//     PlcTask Inputs/GVL_iXlinker.EtherCAT_Master_EJxxxx.Beckhoff_EJ3xxx.A_0005_EJ3058_0000_0020.AI_Standard_Channel_3.Status/Limit_2 <-> AI Standard Channel 3/Status/Limit 2
//     PlcTask Inputs/GVL_iXlinker.EtherCAT_Master_EJxxxx.Beckhoff_EJ3xxx.A_0005_EJ3058_0000_0020.AI_Standard_Channel_4.Status/Limit_1 <-> AI Standard Channel 4/Status/Limit 1
//     PlcTask Inputs/GVL_iXlinker.EtherCAT_Master_EJxxxx.Beckhoff_EJ3xxx.A_0005_EJ3058_0000_0020.AI_Standard_Channel_4.Status/Limit_2 <-> AI Standard Channel 4/Status/Limit 2
//     PlcTask Inputs/GVL_iXlinker.EtherCAT_Master_EJxxxx.Beckhoff_EJ3xxx.A_0005_EJ3058_0000_0020.AI_Standard_Channel_5.Status/Limit_1 <-> AI Standard Channel 5/Status/Limit 1
//     PlcTask Inputs/GVL_iXlinker.EtherCAT_Master_EJxxxx.Beckhoff_EJ3xxx.A_0005_EJ3058_0000_0020.AI_Standard_Channel_5.Status/Limit_2 <-> AI Standard Channel 5/Status/Limit 2
//     PlcTask Inputs/GVL_iXlinker.EtherCAT_Master_EJxxxx.Beckhoff_EJ3xxx.A_0005_EJ3058_0000_0020.AI_Standard_Channel_6.Status/Limit_1 <-> AI Standard Channel 6/Status/Limit 1
//     PlcTask Inputs/GVL_iXlinker.EtherCAT_Master_EJxxxx.Beckhoff_EJ3xxx.A_0005_EJ3058_0000_0020.AI_Standard_Channel_6.Status/Limit_2 <-> AI Standard Channel 6/Status/Limit 2
//     PlcTask Inputs/GVL_iXlinker.EtherCAT_Master_EJxxxx.Beckhoff_EJ3xxx.A_0005_EJ3058_0000_0020.AI_Standard_Channel_7.Status/Limit_1 <-> AI Standard Channel 7/Status/Limit 1
//     PlcTask Inputs/GVL_iXlinker.EtherCAT_Master_EJxxxx.Beckhoff_EJ3xxx.A_0005_EJ3058_0000_0020.AI_Standard_Channel_7.Status/Limit_2 <-> AI Standard Channel 7/Status/Limit 2
//     PlcTask Inputs/GVL_iXlinker.EtherCAT_Master_EJxxxx.Beckhoff_EJ3xxx.A_0005_EJ3058_0000_0020.AI_Standard_Channel_8.Status/Limit_1 <-> AI Standard Channel 8/Status/Limit 1
//     PlcTask Inputs/GVL_iXlinker.EtherCAT_Master_EJxxxx.Beckhoff_EJ3xxx.A_0005_EJ3058_0000_0020.AI_Standard_Channel_8.Status/Limit_2 <-> AI Standard Channel 8/Status/Limit 2
//     PlcTask Inputs/GVL_iXlinker.EtherCAT_Master_EJxxxx.Beckhoff_EJ3xxx.A_0005_EJ3058_0000_0020.AI_Standard_Channel_1.Status/Error <-> AI Standard Channel 1/Status/Error
//     PlcTask Inputs/GVL_iXlinker.EtherCAT_Master_EJxxxx.Beckhoff_EJ3xxx.A_0005_EJ3058_0000_0020.AI_Standard_Channel_2.Status/Error <-> AI Standard Channel 2/Status/Error
//     PlcTask Inputs/GVL_iXlinker.EtherCAT_Master_EJxxxx.Beckhoff_EJ3xxx.A_0005_EJ3058_0000_0020.AI_Standard_Channel_3.Status/Error <-> AI Standard Channel 3/Status/Error
//     PlcTask Inputs/GVL_iXlinker.EtherCAT_Master_EJxxxx.Beckhoff_EJ3xxx.A_0005_EJ3058_0000_0020.AI_Standard_Channel_4.Status/Error <-> AI Standard Channel 4/Status/Error
//     PlcTask Inputs/GVL_iXlinker.EtherCAT_Master_EJxxxx.Beckhoff_EJ3xxx.A_0005_EJ3058_0000_0020.AI_Standard_Channel_5.Status/Error <-> AI Standard Channel 5/Status/Error
//     PlcTask Inputs/GVL_iXlinker.EtherCAT_Master_EJxxxx.Beckhoff_EJ3xxx.A_0005_EJ3058_0000_0020.AI_Standard_Channel_6.Status/Error <-> AI Standard Channel 6/Status/Error
//     PlcTask Inputs/GVL_iXlinker.EtherCAT_Master_EJxxxx.Beckhoff_EJ3xxx.A_0005_EJ3058_0000_0020.AI_Standard_Channel_7.Status/Error <-> AI Standard Channel 7/Status/Error
//     PlcTask Inputs/GVL_iXlinker.EtherCAT_Master_EJxxxx.Beckhoff_EJ3xxx.A_0005_EJ3058_0000_0020.AI_Standard_Channel_8.Status/Error <-> AI Standard Channel 8/Status/Error
//     PlcTask Inputs/GVL_iXlinker.EtherCAT_Master_EJxxxx.Beckhoff_EJ3xxx.A_0005_EJ3058_0000_0020.AI_Standard_Channel_1.Status/TxPDO_State <-> AI Standard Channel 1/Status/TxPDO State
//     PlcTask Inputs/GVL_iXlinker.EtherCAT_Master_EJxxxx.Beckhoff_EJ3xxx.A_0005_EJ3058_0000_0020.AI_Standard_Channel_2.Status/TxPDO_State <-> AI Standard Channel 2/Status/TxPDO State
//     PlcTask Inputs/GVL_iXlinker.EtherCAT_Master_EJxxxx.Beckhoff_EJ3xxx.A_0005_EJ3058_0000_0020.AI_Standard_Channel_3.Status/TxPDO_State <-> AI Standard Channel 3/Status/TxPDO State
//     PlcTask Inputs/GVL_iXlinker.EtherCAT_Master_EJxxxx.Beckhoff_EJ3xxx.A_0005_EJ3058_0000_0020.AI_Standard_Channel_4.Status/TxPDO_State <-> AI Standard Channel 4/Status/TxPDO State
//     PlcTask Inputs/GVL_iXlinker.EtherCAT_Master_EJxxxx.Beckhoff_EJ3xxx.A_0005_EJ3058_0000_0020.AI_Standard_Channel_5.Status/TxPDO_State <-> AI Standard Channel 5/Status/TxPDO State
//     PlcTask Inputs/GVL_iXlinker.EtherCAT_Master_EJxxxx.Beckhoff_EJ3xxx.A_0005_EJ3058_0000_0020.AI_Standard_Channel_6.Status/TxPDO_State <-> AI Standard Channel 6/Status/TxPDO State
//     PlcTask Inputs/GVL_iXlinker.EtherCAT_Master_EJxxxx.Beckhoff_EJ3xxx.A_0005_EJ3058_0000_0020.AI_Standard_Channel_7.Status/TxPDO_State <-> AI Standard Channel 7/Status/TxPDO State
//     PlcTask Inputs/GVL_iXlinker.EtherCAT_Master_EJxxxx.Beckhoff_EJ3xxx.A_0005_EJ3058_0000_0020.AI_Standard_Channel_8.Status/TxPDO_State <-> AI Standard Channel 8/Status/TxPDO State
//     PlcTask Inputs/GVL_iXlinker.EtherCAT_Master_EJxxxx.Beckhoff_EJ3xxx.A_0005_EJ3058_0000_0020.AI_Standard_Channel_1.Status/TxPDO_Toggle <-> AI Standard Channel 1/Status/TxPDO Toggle
//     PlcTask Inputs/GVL_iXlinker.EtherCAT_Master_EJxxxx.Beckhoff_EJ3xxx.A_0005_EJ3058_0000_0020.AI_Standard_Channel_2.Status/TxPDO_Toggle <-> AI Standard Channel 2/Status/TxPDO Toggle
//     PlcTask Inputs/GVL_iXlinker.EtherCAT_Master_EJxxxx.Beckhoff_EJ3xxx.A_0005_EJ3058_0000_0020.AI_Standard_Channel_3.Status/TxPDO_Toggle <-> AI Standard Channel 3/Status/TxPDO Toggle
//     PlcTask Inputs/GVL_iXlinker.EtherCAT_Master_EJxxxx.Beckhoff_EJ3xxx.A_0005_EJ3058_0000_0020.AI_Standard_Channel_4.Status/TxPDO_Toggle <-> AI Standard Channel 4/Status/TxPDO Toggle
//     PlcTask Inputs/GVL_iXlinker.EtherCAT_Master_EJxxxx.Beckhoff_EJ3xxx.A_0005_EJ3058_0000_0020.AI_Standard_Channel_5.Status/TxPDO_Toggle <-> AI Standard Channel 5/Status/TxPDO Toggle
//     PlcTask Inputs/GVL_iXlinker.EtherCAT_Master_EJxxxx.Beckhoff_EJ3xxx.A_0005_EJ3058_0000_0020.AI_Standard_Channel_6.Status/TxPDO_Toggle <-> AI Standard Channel 6/Status/TxPDO Toggle
//     PlcTask Inputs/GVL_iXlinker.EtherCAT_Master_EJxxxx.Beckhoff_EJ3xxx.A_0005_EJ3058_0000_0020.AI_Standard_Channel_7.Status/TxPDO_Toggle <-> AI Standard Channel 7/Status/TxPDO Toggle
//     PlcTask Inputs/GVL_iXlinker.EtherCAT_Master_EJxxxx.Beckhoff_EJ3xxx.A_0005_EJ3058_0000_0020.AI_Standard_Channel_8.Status/TxPDO_Toggle <-> AI Standard Channel 8/Status/TxPDO Toggle
//     PlcTask Inputs/GVL_iXlinker.EtherCAT_Master_EJxxxx.Beckhoff_EJ3xxx.A_0005_EJ3058_0000_0020.AI_Standard_Channel_1.Value <-> AI Standard Channel 1/Value
//     PlcTask Inputs/GVL_iXlinker.EtherCAT_Master_EJxxxx.Beckhoff_EJ3xxx.A_0005_EJ3058_0000_0020.AI_Standard_Channel_2.Value <-> AI Standard Channel 2/Value
//     PlcTask Inputs/GVL_iXlinker.EtherCAT_Master_EJxxxx.Beckhoff_EJ3xxx.A_0005_EJ3058_0000_0020.AI_Standard_Channel_3.Value <-> AI Standard Channel 3/Value
//     PlcTask Inputs/GVL_iXlinker.EtherCAT_Master_EJxxxx.Beckhoff_EJ3xxx.A_0005_EJ3058_0000_0020.AI_Standard_Channel_4.Value <-> AI Standard Channel 4/Value
//     PlcTask Inputs/GVL_iXlinker.EtherCAT_Master_EJxxxx.Beckhoff_EJ3xxx.A_0005_EJ3058_0000_0020.AI_Standard_Channel_5.Value <-> AI Standard Channel 5/Value
//     PlcTask Inputs/GVL_iXlinker.EtherCAT_Master_EJxxxx.Beckhoff_EJ3xxx.A_0005_EJ3058_0000_0020.AI_Standard_Channel_6.Value <-> AI Standard Channel 6/Value
//     PlcTask Inputs/GVL_iXlinker.EtherCAT_Master_EJxxxx.Beckhoff_EJ3xxx.A_0005_EJ3058_0000_0020.AI_Standard_Channel_7.Value <-> AI Standard Channel 7/Value
//     PlcTask Inputs/GVL_iXlinker.EtherCAT_Master_EJxxxx.Beckhoff_EJ3xxx.A_0005_EJ3058_0000_0020.AI_Standard_Channel_8.Value <-> AI Standard Channel 8/Value
//     PlcTask Inputs/GVL_iXlinker.EtherCAT_Master_EJxxxx.Beckhoff_EJ3xxx.A_0005_EJ3058_0000_0020.WcState.WcState <-> WcState/WcState
//     PlcTask Inputs/GVL_iXlinker.EtherCAT_Master_EJxxxx.Beckhoff_EJ3xxx.A_0005_EJ3058_0000_0020.WcState.InputToggle <-> WcState/InputToggle
//     PlcTask Inputs/GVL_iXlinker.EtherCAT_Master_EJxxxx.Beckhoff_EJ3xxx.A_0005_EJ3058_0000_0020.InfoData.AdsAddr <-> InfoData/AdsAddr
//     PlcTask Inputs/GVL_iXlinker.EtherCAT_Master_EJxxxx.Beckhoff_EJ3xxx.A_0005_EJ3058_0000_0020.InfoData.State <-> InfoData/State
//   PLC/PLC Instance <-> EtherCAT Master EJxxxx/Beckhoff EJ3xxx/A_0006(EJ3068-0000-0020)
//     PlcTask Inputs/GVL_iXlinker.EtherCAT_Master_EJxxxx.Beckhoff_EJ3xxx.A_0006_EJ3068_0000_0020.AI_Standard_Channel_1.Status/Underrange <-> AI Standard Channel 1/Status/Underrange
//     PlcTask Inputs/GVL_iXlinker.EtherCAT_Master_EJxxxx.Beckhoff_EJ3xxx.A_0006_EJ3068_0000_0020.AI_Standard_Channel_2.Status/Underrange <-> AI Standard Channel 2/Status/Underrange
//     PlcTask Inputs/GVL_iXlinker.EtherCAT_Master_EJxxxx.Beckhoff_EJ3xxx.A_0006_EJ3068_0000_0020.AI_Standard_Channel_3.Status/Underrange <-> AI Standard Channel 3/Status/Underrange
//     PlcTask Inputs/GVL_iXlinker.EtherCAT_Master_EJxxxx.Beckhoff_EJ3xxx.A_0006_EJ3068_0000_0020.AI_Standard_Channel_4.Status/Underrange <-> AI Standard Channel 4/Status/Underrange
//     PlcTask Inputs/GVL_iXlinker.EtherCAT_Master_EJxxxx.Beckhoff_EJ3xxx.A_0006_EJ3068_0000_0020.AI_Standard_Channel_5.Status/Underrange <-> AI Standard Channel 5/Status/Underrange
//     PlcTask Inputs/GVL_iXlinker.EtherCAT_Master_EJxxxx.Beckhoff_EJ3xxx.A_0006_EJ3068_0000_0020.AI_Standard_Channel_6.Status/Underrange <-> AI Standard Channel 6/Status/Underrange
//     PlcTask Inputs/GVL_iXlinker.EtherCAT_Master_EJxxxx.Beckhoff_EJ3xxx.A_0006_EJ3068_0000_0020.AI_Standard_Channel_7.Status/Underrange <-> AI Standard Channel 7/Status/Underrange
//     PlcTask Inputs/GVL_iXlinker.EtherCAT_Master_EJxxxx.Beckhoff_EJ3xxx.A_0006_EJ3068_0000_0020.AI_Standard_Channel_8.Status/Underrange <-> AI Standard Channel 8/Status/Underrange
//     PlcTask Inputs/GVL_iXlinker.EtherCAT_Master_EJxxxx.Beckhoff_EJ3xxx.A_0006_EJ3068_0000_0020.AI_Standard_Channel_1.Status/Overrange <-> AI Standard Channel 1/Status/Overrange
//     PlcTask Inputs/GVL_iXlinker.EtherCAT_Master_EJxxxx.Beckhoff_EJ3xxx.A_0006_EJ3068_0000_0020.AI_Standard_Channel_2.Status/Overrange <-> AI Standard Channel 2/Status/Overrange
//     PlcTask Inputs/GVL_iXlinker.EtherCAT_Master_EJxxxx.Beckhoff_EJ3xxx.A_0006_EJ3068_0000_0020.AI_Standard_Channel_3.Status/Overrange <-> AI Standard Channel 3/Status/Overrange
//     PlcTask Inputs/GVL_iXlinker.EtherCAT_Master_EJxxxx.Beckhoff_EJ3xxx.A_0006_EJ3068_0000_0020.AI_Standard_Channel_4.Status/Overrange <-> AI Standard Channel 4/Status/Overrange
//     PlcTask Inputs/GVL_iXlinker.EtherCAT_Master_EJxxxx.Beckhoff_EJ3xxx.A_0006_EJ3068_0000_0020.AI_Standard_Channel_5.Status/Overrange <-> AI Standard Channel 5/Status/Overrange
//     PlcTask Inputs/GVL_iXlinker.EtherCAT_Master_EJxxxx.Beckhoff_EJ3xxx.A_0006_EJ3068_0000_0020.AI_Standard_Channel_6.Status/Overrange <-> AI Standard Channel 6/Status/Overrange
//     PlcTask Inputs/GVL_iXlinker.EtherCAT_Master_EJxxxx.Beckhoff_EJ3xxx.A_0006_EJ3068_0000_0020.AI_Standard_Channel_7.Status/Overrange <-> AI Standard Channel 7/Status/Overrange
//     PlcTask Inputs/GVL_iXlinker.EtherCAT_Master_EJxxxx.Beckhoff_EJ3xxx.A_0006_EJ3068_0000_0020.AI_Standard_Channel_8.Status/Overrange <-> AI Standard Channel 8/Status/Overrange
//     PlcTask Inputs/GVL_iXlinker.EtherCAT_Master_EJxxxx.Beckhoff_EJ3xxx.A_0006_EJ3068_0000_0020.AI_Standard_Channel_1.Status/Limit_1 <-> AI Standard Channel 1/Status/Limit 1
//     PlcTask Inputs/GVL_iXlinker.EtherCAT_Master_EJxxxx.Beckhoff_EJ3xxx.A_0006_EJ3068_0000_0020.AI_Standard_Channel_1.Status/Limit_2 <-> AI Standard Channel 1/Status/Limit 2
//     PlcTask Inputs/GVL_iXlinker.EtherCAT_Master_EJxxxx.Beckhoff_EJ3xxx.A_0006_EJ3068_0000_0020.AI_Standard_Channel_2.Status/Limit_1 <-> AI Standard Channel 2/Status/Limit 1
//     PlcTask Inputs/GVL_iXlinker.EtherCAT_Master_EJxxxx.Beckhoff_EJ3xxx.A_0006_EJ3068_0000_0020.AI_Standard_Channel_2.Status/Limit_2 <-> AI Standard Channel 2/Status/Limit 2
//     PlcTask Inputs/GVL_iXlinker.EtherCAT_Master_EJxxxx.Beckhoff_EJ3xxx.A_0006_EJ3068_0000_0020.AI_Standard_Channel_3.Status/Limit_1 <-> AI Standard Channel 3/Status/Limit 1
//     PlcTask Inputs/GVL_iXlinker.EtherCAT_Master_EJxxxx.Beckhoff_EJ3xxx.A_0006_EJ3068_0000_0020.AI_Standard_Channel_3.Status/Limit_2 <-> AI Standard Channel 3/Status/Limit 2
//     PlcTask Inputs/GVL_iXlinker.EtherCAT_Master_EJxxxx.Beckhoff_EJ3xxx.A_0006_EJ3068_0000_0020.AI_Standard_Channel_4.Status/Limit_1 <-> AI Standard Channel 4/Status/Limit 1
//     PlcTask Inputs/GVL_iXlinker.EtherCAT_Master_EJxxxx.Beckhoff_EJ3xxx.A_0006_EJ3068_0000_0020.AI_Standard_Channel_4.Status/Limit_2 <-> AI Standard Channel 4/Status/Limit 2
//     PlcTask Inputs/GVL_iXlinker.EtherCAT_Master_EJxxxx.Beckhoff_EJ3xxx.A_0006_EJ3068_0000_0020.AI_Standard_Channel_5.Status/Limit_1 <-> AI Standard Channel 5/Status/Limit 1
//     PlcTask Inputs/GVL_iXlinker.EtherCAT_Master_EJxxxx.Beckhoff_EJ3xxx.A_0006_EJ3068_0000_0020.AI_Standard_Channel_5.Status/Limit_2 <-> AI Standard Channel 5/Status/Limit 2
//     PlcTask Inputs/GVL_iXlinker.EtherCAT_Master_EJxxxx.Beckhoff_EJ3xxx.A_0006_EJ3068_0000_0020.AI_Standard_Channel_6.Status/Limit_1 <-> AI Standard Channel 6/Status/Limit 1
//     PlcTask Inputs/GVL_iXlinker.EtherCAT_Master_EJxxxx.Beckhoff_EJ3xxx.A_0006_EJ3068_0000_0020.AI_Standard_Channel_6.Status/Limit_2 <-> AI Standard Channel 6/Status/Limit 2
//     PlcTask Inputs/GVL_iXlinker.EtherCAT_Master_EJxxxx.Beckhoff_EJ3xxx.A_0006_EJ3068_0000_0020.AI_Standard_Channel_7.Status/Limit_1 <-> AI Standard Channel 7/Status/Limit 1
//     PlcTask Inputs/GVL_iXlinker.EtherCAT_Master_EJxxxx.Beckhoff_EJ3xxx.A_0006_EJ3068_0000_0020.AI_Standard_Channel_7.Status/Limit_2 <-> AI Standard Channel 7/Status/Limit 2
//     PlcTask Inputs/GVL_iXlinker.EtherCAT_Master_EJxxxx.Beckhoff_EJ3xxx.A_0006_EJ3068_0000_0020.AI_Standard_Channel_8.Status/Limit_1 <-> AI Standard Channel 8/Status/Limit 1
//     PlcTask Inputs/GVL_iXlinker.EtherCAT_Master_EJxxxx.Beckhoff_EJ3xxx.A_0006_EJ3068_0000_0020.AI_Standard_Channel_8.Status/Limit_2 <-> AI Standard Channel 8/Status/Limit 2
//     PlcTask Inputs/GVL_iXlinker.EtherCAT_Master_EJxxxx.Beckhoff_EJ3xxx.A_0006_EJ3068_0000_0020.AI_Standard_Channel_1.Status/Error <-> AI Standard Channel 1/Status/Error
//     PlcTask Inputs/GVL_iXlinker.EtherCAT_Master_EJxxxx.Beckhoff_EJ3xxx.A_0006_EJ3068_0000_0020.AI_Standard_Channel_2.Status/Error <-> AI Standard Channel 2/Status/Error
//     PlcTask Inputs/GVL_iXlinker.EtherCAT_Master_EJxxxx.Beckhoff_EJ3xxx.A_0006_EJ3068_0000_0020.AI_Standard_Channel_3.Status/Error <-> AI Standard Channel 3/Status/Error
//     PlcTask Inputs/GVL_iXlinker.EtherCAT_Master_EJxxxx.Beckhoff_EJ3xxx.A_0006_EJ3068_0000_0020.AI_Standard_Channel_4.Status/Error <-> AI Standard Channel 4/Status/Error
//     PlcTask Inputs/GVL_iXlinker.EtherCAT_Master_EJxxxx.Beckhoff_EJ3xxx.A_0006_EJ3068_0000_0020.AI_Standard_Channel_5.Status/Error <-> AI Standard Channel 5/Status/Error
//     PlcTask Inputs/GVL_iXlinker.EtherCAT_Master_EJxxxx.Beckhoff_EJ3xxx.A_0006_EJ3068_0000_0020.AI_Standard_Channel_6.Status/Error <-> AI Standard Channel 6/Status/Error
//     PlcTask Inputs/GVL_iXlinker.EtherCAT_Master_EJxxxx.Beckhoff_EJ3xxx.A_0006_EJ3068_0000_0020.AI_Standard_Channel_7.Status/Error <-> AI Standard Channel 7/Status/Error
//     PlcTask Inputs/GVL_iXlinker.EtherCAT_Master_EJxxxx.Beckhoff_EJ3xxx.A_0006_EJ3068_0000_0020.AI_Standard_Channel_8.Status/Error <-> AI Standard Channel 8/Status/Error
//     PlcTask Inputs/GVL_iXlinker.EtherCAT_Master_EJxxxx.Beckhoff_EJ3xxx.A_0006_EJ3068_0000_0020.AI_Standard_Channel_1.Status/TxPDO_State <-> AI Standard Channel 1/Status/TxPDO State
//     PlcTask Inputs/GVL_iXlinker.EtherCAT_Master_EJxxxx.Beckhoff_EJ3xxx.A_0006_EJ3068_0000_0020.AI_Standard_Channel_2.Status/TxPDO_State <-> AI Standard Channel 2/Status/TxPDO State
//     PlcTask Inputs/GVL_iXlinker.EtherCAT_Master_EJxxxx.Beckhoff_EJ3xxx.A_0006_EJ3068_0000_0020.AI_Standard_Channel_3.Status/TxPDO_State <-> AI Standard Channel 3/Status/TxPDO State
//     PlcTask Inputs/GVL_iXlinker.EtherCAT_Master_EJxxxx.Beckhoff_EJ3xxx.A_0006_EJ3068_0000_0020.AI_Standard_Channel_4.Status/TxPDO_State <-> AI Standard Channel 4/Status/TxPDO State
//     PlcTask Inputs/GVL_iXlinker.EtherCAT_Master_EJxxxx.Beckhoff_EJ3xxx.A_0006_EJ3068_0000_0020.AI_Standard_Channel_5.Status/TxPDO_State <-> AI Standard Channel 5/Status/TxPDO State
//     PlcTask Inputs/GVL_iXlinker.EtherCAT_Master_EJxxxx.Beckhoff_EJ3xxx.A_0006_EJ3068_0000_0020.AI_Standard_Channel_6.Status/TxPDO_State <-> AI Standard Channel 6/Status/TxPDO State
//     PlcTask Inputs/GVL_iXlinker.EtherCAT_Master_EJxxxx.Beckhoff_EJ3xxx.A_0006_EJ3068_0000_0020.AI_Standard_Channel_7.Status/TxPDO_State <-> AI Standard Channel 7/Status/TxPDO State
//     PlcTask Inputs/GVL_iXlinker.EtherCAT_Master_EJxxxx.Beckhoff_EJ3xxx.A_0006_EJ3068_0000_0020.AI_Standard_Channel_8.Status/TxPDO_State <-> AI Standard Channel 8/Status/TxPDO State
//     PlcTask Inputs/GVL_iXlinker.EtherCAT_Master_EJxxxx.Beckhoff_EJ3xxx.A_0006_EJ3068_0000_0020.AI_Standard_Channel_1.Status/TxPDO_Toggle <-> AI Standard Channel 1/Status/TxPDO Toggle
//     PlcTask Inputs/GVL_iXlinker.EtherCAT_Master_EJxxxx.Beckhoff_EJ3xxx.A_0006_EJ3068_0000_0020.AI_Standard_Channel_2.Status/TxPDO_Toggle <-> AI Standard Channel 2/Status/TxPDO Toggle
//     PlcTask Inputs/GVL_iXlinker.EtherCAT_Master_EJxxxx.Beckhoff_EJ3xxx.A_0006_EJ3068_0000_0020.AI_Standard_Channel_3.Status/TxPDO_Toggle <-> AI Standard Channel 3/Status/TxPDO Toggle
//     PlcTask Inputs/GVL_iXlinker.EtherCAT_Master_EJxxxx.Beckhoff_EJ3xxx.A_0006_EJ3068_0000_0020.AI_Standard_Channel_4.Status/TxPDO_Toggle <-> AI Standard Channel 4/Status/TxPDO Toggle
//     PlcTask Inputs/GVL_iXlinker.EtherCAT_Master_EJxxxx.Beckhoff_EJ3xxx.A_0006_EJ3068_0000_0020.AI_Standard_Channel_5.Status/TxPDO_Toggle <-> AI Standard Channel 5/Status/TxPDO Toggle
//     PlcTask Inputs/GVL_iXlinker.EtherCAT_Master_EJxxxx.Beckhoff_EJ3xxx.A_0006_EJ3068_0000_0020.AI_Standard_Channel_6.Status/TxPDO_Toggle <-> AI Standard Channel 6/Status/TxPDO Toggle
//     PlcTask Inputs/GVL_iXlinker.EtherCAT_Master_EJxxxx.Beckhoff_EJ3xxx.A_0006_EJ3068_0000_0020.AI_Standard_Channel_7.Status/TxPDO_Toggle <-> AI Standard Channel 7/Status/TxPDO Toggle
//     PlcTask Inputs/GVL_iXlinker.EtherCAT_Master_EJxxxx.Beckhoff_EJ3xxx.A_0006_EJ3068_0000_0020.AI_Standard_Channel_8.Status/TxPDO_Toggle <-> AI Standard Channel 8/Status/TxPDO Toggle
//     PlcTask Inputs/GVL_iXlinker.EtherCAT_Master_EJxxxx.Beckhoff_EJ3xxx.A_0006_EJ3068_0000_0020.AI_Standard_Channel_1.Value <-> AI Standard Channel 1/Value
//     PlcTask Inputs/GVL_iXlinker.EtherCAT_Master_EJxxxx.Beckhoff_EJ3xxx.A_0006_EJ3068_0000_0020.AI_Standard_Channel_2.Value <-> AI Standard Channel 2/Value
//     PlcTask Inputs/GVL_iXlinker.EtherCAT_Master_EJxxxx.Beckhoff_EJ3xxx.A_0006_EJ3068_0000_0020.AI_Standard_Channel_3.Value <-> AI Standard Channel 3/Value
//     PlcTask Inputs/GVL_iXlinker.EtherCAT_Master_EJxxxx.Beckhoff_EJ3xxx.A_0006_EJ3068_0000_0020.AI_Standard_Channel_4.Value <-> AI Standard Channel 4/Value
//     PlcTask Inputs/GVL_iXlinker.EtherCAT_Master_EJxxxx.Beckhoff_EJ3xxx.A_0006_EJ3068_0000_0020.AI_Standard_Channel_5.Value <-> AI Standard Channel 5/Value
//     PlcTask Inputs/GVL_iXlinker.EtherCAT_Master_EJxxxx.Beckhoff_EJ3xxx.A_0006_EJ3068_0000_0020.AI_Standard_Channel_6.Value <-> AI Standard Channel 6/Value
//     PlcTask Inputs/GVL_iXlinker.EtherCAT_Master_EJxxxx.Beckhoff_EJ3xxx.A_0006_EJ3068_0000_0020.AI_Standard_Channel_7.Value <-> AI Standard Channel 7/Value
//     PlcTask Inputs/GVL_iXlinker.EtherCAT_Master_EJxxxx.Beckhoff_EJ3xxx.A_0006_EJ3068_0000_0020.AI_Standard_Channel_8.Value <-> AI Standard Channel 8/Value
//     PlcTask Inputs/GVL_iXlinker.EtherCAT_Master_EJxxxx.Beckhoff_EJ3xxx.A_0006_EJ3068_0000_0020.WcState.WcState <-> WcState/WcState
//     PlcTask Inputs/GVL_iXlinker.EtherCAT_Master_EJxxxx.Beckhoff_EJ3xxx.A_0006_EJ3068_0000_0020.WcState.InputToggle <-> WcState/InputToggle
//     PlcTask Inputs/GVL_iXlinker.EtherCAT_Master_EJxxxx.Beckhoff_EJ3xxx.A_0006_EJ3068_0000_0020.InfoData.AdsAddr <-> InfoData/AdsAddr
//     PlcTask Inputs/GVL_iXlinker.EtherCAT_Master_EJxxxx.Beckhoff_EJ3xxx.A_0006_EJ3068_0000_0020.InfoData.State <-> InfoData/State
//   PLC/PLC Instance <-> EtherCAT Master EJxxxx/Beckhoff EJ3xxx/A_0007(EJ3068-0000-0021)
//     PlcTask Inputs/GVL_iXlinker.EtherCAT_Master_EJxxxx.Beckhoff_EJ3xxx.A_0007_EJ3068_0000_0021.AI_Standard_Channel_1.Status/Underrange <-> AI Standard Channel 1/Status/Underrange
//     PlcTask Inputs/GVL_iXlinker.EtherCAT_Master_EJxxxx.Beckhoff_EJ3xxx.A_0007_EJ3068_0000_0021.AI_Standard_Channel_2.Status/Underrange <-> AI Standard Channel 2/Status/Underrange
//     PlcTask Inputs/GVL_iXlinker.EtherCAT_Master_EJxxxx.Beckhoff_EJ3xxx.A_0007_EJ3068_0000_0021.AI_Standard_Channel_3.Status/Underrange <-> AI Standard Channel 3/Status/Underrange
//     PlcTask Inputs/GVL_iXlinker.EtherCAT_Master_EJxxxx.Beckhoff_EJ3xxx.A_0007_EJ3068_0000_0021.AI_Standard_Channel_4.Status/Underrange <-> AI Standard Channel 4/Status/Underrange
//     PlcTask Inputs/GVL_iXlinker.EtherCAT_Master_EJxxxx.Beckhoff_EJ3xxx.A_0007_EJ3068_0000_0021.AI_Standard_Channel_5.Status/Underrange <-> AI Standard Channel 5/Status/Underrange
//     PlcTask Inputs/GVL_iXlinker.EtherCAT_Master_EJxxxx.Beckhoff_EJ3xxx.A_0007_EJ3068_0000_0021.AI_Standard_Channel_6.Status/Underrange <-> AI Standard Channel 6/Status/Underrange
//     PlcTask Inputs/GVL_iXlinker.EtherCAT_Master_EJxxxx.Beckhoff_EJ3xxx.A_0007_EJ3068_0000_0021.AI_Standard_Channel_7.Status/Underrange <-> AI Standard Channel 7/Status/Underrange
//     PlcTask Inputs/GVL_iXlinker.EtherCAT_Master_EJxxxx.Beckhoff_EJ3xxx.A_0007_EJ3068_0000_0021.AI_Standard_Channel_8.Status/Underrange <-> AI Standard Channel 8/Status/Underrange
//     PlcTask Inputs/GVL_iXlinker.EtherCAT_Master_EJxxxx.Beckhoff_EJ3xxx.A_0007_EJ3068_0000_0021.AI_Standard_Channel_1.Status/Overrange <-> AI Standard Channel 1/Status/Overrange
//     PlcTask Inputs/GVL_iXlinker.EtherCAT_Master_EJxxxx.Beckhoff_EJ3xxx.A_0007_EJ3068_0000_0021.AI_Standard_Channel_2.Status/Overrange <-> AI Standard Channel 2/Status/Overrange
//     PlcTask Inputs/GVL_iXlinker.EtherCAT_Master_EJxxxx.Beckhoff_EJ3xxx.A_0007_EJ3068_0000_0021.AI_Standard_Channel_3.Status/Overrange <-> AI Standard Channel 3/Status/Overrange
//     PlcTask Inputs/GVL_iXlinker.EtherCAT_Master_EJxxxx.Beckhoff_EJ3xxx.A_0007_EJ3068_0000_0021.AI_Standard_Channel_4.Status/Overrange <-> AI Standard Channel 4/Status/Overrange
//     PlcTask Inputs/GVL_iXlinker.EtherCAT_Master_EJxxxx.Beckhoff_EJ3xxx.A_0007_EJ3068_0000_0021.AI_Standard_Channel_5.Status/Overrange <-> AI Standard Channel 5/Status/Overrange
//     PlcTask Inputs/GVL_iXlinker.EtherCAT_Master_EJxxxx.Beckhoff_EJ3xxx.A_0007_EJ3068_0000_0021.AI_Standard_Channel_6.Status/Overrange <-> AI Standard Channel 6/Status/Overrange
//     PlcTask Inputs/GVL_iXlinker.EtherCAT_Master_EJxxxx.Beckhoff_EJ3xxx.A_0007_EJ3068_0000_0021.AI_Standard_Channel_7.Status/Overrange <-> AI Standard Channel 7/Status/Overrange
//     PlcTask Inputs/GVL_iXlinker.EtherCAT_Master_EJxxxx.Beckhoff_EJ3xxx.A_0007_EJ3068_0000_0021.AI_Standard_Channel_8.Status/Overrange <-> AI Standard Channel 8/Status/Overrange
//     PlcTask Inputs/GVL_iXlinker.EtherCAT_Master_EJxxxx.Beckhoff_EJ3xxx.A_0007_EJ3068_0000_0021.AI_Standard_Channel_1.Status/Limit_1 <-> AI Standard Channel 1/Status/Limit 1
//     PlcTask Inputs/GVL_iXlinker.EtherCAT_Master_EJxxxx.Beckhoff_EJ3xxx.A_0007_EJ3068_0000_0021.AI_Standard_Channel_1.Status/Limit_2 <-> AI Standard Channel 1/Status/Limit 2
//     PlcTask Inputs/GVL_iXlinker.EtherCAT_Master_EJxxxx.Beckhoff_EJ3xxx.A_0007_EJ3068_0000_0021.AI_Standard_Channel_2.Status/Limit_1 <-> AI Standard Channel 2/Status/Limit 1
//     PlcTask Inputs/GVL_iXlinker.EtherCAT_Master_EJxxxx.Beckhoff_EJ3xxx.A_0007_EJ3068_0000_0021.AI_Standard_Channel_2.Status/Limit_2 <-> AI Standard Channel 2/Status/Limit 2
//     PlcTask Inputs/GVL_iXlinker.EtherCAT_Master_EJxxxx.Beckhoff_EJ3xxx.A_0007_EJ3068_0000_0021.AI_Standard_Channel_3.Status/Limit_1 <-> AI Standard Channel 3/Status/Limit 1
//     PlcTask Inputs/GVL_iXlinker.EtherCAT_Master_EJxxxx.Beckhoff_EJ3xxx.A_0007_EJ3068_0000_0021.AI_Standard_Channel_3.Status/Limit_2 <-> AI Standard Channel 3/Status/Limit 2
//     PlcTask Inputs/GVL_iXlinker.EtherCAT_Master_EJxxxx.Beckhoff_EJ3xxx.A_0007_EJ3068_0000_0021.AI_Standard_Channel_4.Status/Limit_1 <-> AI Standard Channel 4/Status/Limit 1
//     PlcTask Inputs/GVL_iXlinker.EtherCAT_Master_EJxxxx.Beckhoff_EJ3xxx.A_0007_EJ3068_0000_0021.AI_Standard_Channel_4.Status/Limit_2 <-> AI Standard Channel 4/Status/Limit 2
//     PlcTask Inputs/GVL_iXlinker.EtherCAT_Master_EJxxxx.Beckhoff_EJ3xxx.A_0007_EJ3068_0000_0021.AI_Standard_Channel_5.Status/Limit_1 <-> AI Standard Channel 5/Status/Limit 1
//     PlcTask Inputs/GVL_iXlinker.EtherCAT_Master_EJxxxx.Beckhoff_EJ3xxx.A_0007_EJ3068_0000_0021.AI_Standard_Channel_5.Status/Limit_2 <-> AI Standard Channel 5/Status/Limit 2
//     PlcTask Inputs/GVL_iXlinker.EtherCAT_Master_EJxxxx.Beckhoff_EJ3xxx.A_0007_EJ3068_0000_0021.AI_Standard_Channel_6.Status/Limit_1 <-> AI Standard Channel 6/Status/Limit 1
//     PlcTask Inputs/GVL_iXlinker.EtherCAT_Master_EJxxxx.Beckhoff_EJ3xxx.A_0007_EJ3068_0000_0021.AI_Standard_Channel_6.Status/Limit_2 <-> AI Standard Channel 6/Status/Limit 2
//     PlcTask Inputs/GVL_iXlinker.EtherCAT_Master_EJxxxx.Beckhoff_EJ3xxx.A_0007_EJ3068_0000_0021.AI_Standard_Channel_7.Status/Limit_1 <-> AI Standard Channel 7/Status/Limit 1
//     PlcTask Inputs/GVL_iXlinker.EtherCAT_Master_EJxxxx.Beckhoff_EJ3xxx.A_0007_EJ3068_0000_0021.AI_Standard_Channel_7.Status/Limit_2 <-> AI Standard Channel 7/Status/Limit 2
//     PlcTask Inputs/GVL_iXlinker.EtherCAT_Master_EJxxxx.Beckhoff_EJ3xxx.A_0007_EJ3068_0000_0021.AI_Standard_Channel_8.Status/Limit_1 <-> AI Standard Channel 8/Status/Limit 1
//     PlcTask Inputs/GVL_iXlinker.EtherCAT_Master_EJxxxx.Beckhoff_EJ3xxx.A_0007_EJ3068_0000_0021.AI_Standard_Channel_8.Status/Limit_2 <-> AI Standard Channel 8/Status/Limit 2
//     PlcTask Inputs/GVL_iXlinker.EtherCAT_Master_EJxxxx.Beckhoff_EJ3xxx.A_0007_EJ3068_0000_0021.AI_Standard_Channel_1.Status/Error <-> AI Standard Channel 1/Status/Error
//     PlcTask Inputs/GVL_iXlinker.EtherCAT_Master_EJxxxx.Beckhoff_EJ3xxx.A_0007_EJ3068_0000_0021.AI_Standard_Channel_2.Status/Error <-> AI Standard Channel 2/Status/Error
//     PlcTask Inputs/GVL_iXlinker.EtherCAT_Master_EJxxxx.Beckhoff_EJ3xxx.A_0007_EJ3068_0000_0021.AI_Standard_Channel_3.Status/Error <-> AI Standard Channel 3/Status/Error
//     PlcTask Inputs/GVL_iXlinker.EtherCAT_Master_EJxxxx.Beckhoff_EJ3xxx.A_0007_EJ3068_0000_0021.AI_Standard_Channel_4.Status/Error <-> AI Standard Channel 4/Status/Error
//     PlcTask Inputs/GVL_iXlinker.EtherCAT_Master_EJxxxx.Beckhoff_EJ3xxx.A_0007_EJ3068_0000_0021.AI_Standard_Channel_5.Status/Error <-> AI Standard Channel 5/Status/Error
//     PlcTask Inputs/GVL_iXlinker.EtherCAT_Master_EJxxxx.Beckhoff_EJ3xxx.A_0007_EJ3068_0000_0021.AI_Standard_Channel_6.Status/Error <-> AI Standard Channel 6/Status/Error
//     PlcTask Inputs/GVL_iXlinker.EtherCAT_Master_EJxxxx.Beckhoff_EJ3xxx.A_0007_EJ3068_0000_0021.AI_Standard_Channel_7.Status/Error <-> AI Standard Channel 7/Status/Error
//     PlcTask Inputs/GVL_iXlinker.EtherCAT_Master_EJxxxx.Beckhoff_EJ3xxx.A_0007_EJ3068_0000_0021.AI_Standard_Channel_8.Status/Error <-> AI Standard Channel 8/Status/Error
//     PlcTask Inputs/GVL_iXlinker.EtherCAT_Master_EJxxxx.Beckhoff_EJ3xxx.A_0007_EJ3068_0000_0021.AI_Standard_Channel_1.Status/TxPDO_State <-> AI Standard Channel 1/Status/TxPDO State
//     PlcTask Inputs/GVL_iXlinker.EtherCAT_Master_EJxxxx.Beckhoff_EJ3xxx.A_0007_EJ3068_0000_0021.AI_Standard_Channel_2.Status/TxPDO_State <-> AI Standard Channel 2/Status/TxPDO State
//     PlcTask Inputs/GVL_iXlinker.EtherCAT_Master_EJxxxx.Beckhoff_EJ3xxx.A_0007_EJ3068_0000_0021.AI_Standard_Channel_3.Status/TxPDO_State <-> AI Standard Channel 3/Status/TxPDO State
//     PlcTask Inputs/GVL_iXlinker.EtherCAT_Master_EJxxxx.Beckhoff_EJ3xxx.A_0007_EJ3068_0000_0021.AI_Standard_Channel_4.Status/TxPDO_State <-> AI Standard Channel 4/Status/TxPDO State
//     PlcTask Inputs/GVL_iXlinker.EtherCAT_Master_EJxxxx.Beckhoff_EJ3xxx.A_0007_EJ3068_0000_0021.AI_Standard_Channel_5.Status/TxPDO_State <-> AI Standard Channel 5/Status/TxPDO State
//     PlcTask Inputs/GVL_iXlinker.EtherCAT_Master_EJxxxx.Beckhoff_EJ3xxx.A_0007_EJ3068_0000_0021.AI_Standard_Channel_6.Status/TxPDO_State <-> AI Standard Channel 6/Status/TxPDO State
//     PlcTask Inputs/GVL_iXlinker.EtherCAT_Master_EJxxxx.Beckhoff_EJ3xxx.A_0007_EJ3068_0000_0021.AI_Standard_Channel_7.Status/TxPDO_State <-> AI Standard Channel 7/Status/TxPDO State
//     PlcTask Inputs/GVL_iXlinker.EtherCAT_Master_EJxxxx.Beckhoff_EJ3xxx.A_0007_EJ3068_0000_0021.AI_Standard_Channel_8.Status/TxPDO_State <-> AI Standard Channel 8/Status/TxPDO State
//     PlcTask Inputs/GVL_iXlinker.EtherCAT_Master_EJxxxx.Beckhoff_EJ3xxx.A_0007_EJ3068_0000_0021.AI_Standard_Channel_1.Status/TxPDO_Toggle <-> AI Standard Channel 1/Status/TxPDO Toggle
//     PlcTask Inputs/GVL_iXlinker.EtherCAT_Master_EJxxxx.Beckhoff_EJ3xxx.A_0007_EJ3068_0000_0021.AI_Standard_Channel_2.Status/TxPDO_Toggle <-> AI Standard Channel 2/Status/TxPDO Toggle
//     PlcTask Inputs/GVL_iXlinker.EtherCAT_Master_EJxxxx.Beckhoff_EJ3xxx.A_0007_EJ3068_0000_0021.AI_Standard_Channel_3.Status/TxPDO_Toggle <-> AI Standard Channel 3/Status/TxPDO Toggle
//     PlcTask Inputs/GVL_iXlinker.EtherCAT_Master_EJxxxx.Beckhoff_EJ3xxx.A_0007_EJ3068_0000_0021.AI_Standard_Channel_4.Status/TxPDO_Toggle <-> AI Standard Channel 4/Status/TxPDO Toggle
//     PlcTask Inputs/GVL_iXlinker.EtherCAT_Master_EJxxxx.Beckhoff_EJ3xxx.A_0007_EJ3068_0000_0021.AI_Standard_Channel_5.Status/TxPDO_Toggle <-> AI Standard Channel 5/Status/TxPDO Toggle
//     PlcTask Inputs/GVL_iXlinker.EtherCAT_Master_EJxxxx.Beckhoff_EJ3xxx.A_0007_EJ3068_0000_0021.AI_Standard_Channel_6.Status/TxPDO_Toggle <-> AI Standard Channel 6/Status/TxPDO Toggle
//     PlcTask Inputs/GVL_iXlinker.EtherCAT_Master_EJxxxx.Beckhoff_EJ3xxx.A_0007_EJ3068_0000_0021.AI_Standard_Channel_7.Status/TxPDO_Toggle <-> AI Standard Channel 7/Status/TxPDO Toggle
//     PlcTask Inputs/GVL_iXlinker.EtherCAT_Master_EJxxxx.Beckhoff_EJ3xxx.A_0007_EJ3068_0000_0021.AI_Standard_Channel_8.Status/TxPDO_Toggle <-> AI Standard Channel 8/Status/TxPDO Toggle
//     PlcTask Inputs/GVL_iXlinker.EtherCAT_Master_EJxxxx.Beckhoff_EJ3xxx.A_0007_EJ3068_0000_0021.AI_Standard_Channel_1.Value <-> AI Standard Channel 1/Value
//     PlcTask Inputs/GVL_iXlinker.EtherCAT_Master_EJxxxx.Beckhoff_EJ3xxx.A_0007_EJ3068_0000_0021.AI_Standard_Channel_2.Value <-> AI Standard Channel 2/Value
//     PlcTask Inputs/GVL_iXlinker.EtherCAT_Master_EJxxxx.Beckhoff_EJ3xxx.A_0007_EJ3068_0000_0021.AI_Standard_Channel_3.Value <-> AI Standard Channel 3/Value
//     PlcTask Inputs/GVL_iXlinker.EtherCAT_Master_EJxxxx.Beckhoff_EJ3xxx.A_0007_EJ3068_0000_0021.AI_Standard_Channel_4.Value <-> AI Standard Channel 4/Value
//     PlcTask Inputs/GVL_iXlinker.EtherCAT_Master_EJxxxx.Beckhoff_EJ3xxx.A_0007_EJ3068_0000_0021.AI_Standard_Channel_5.Value <-> AI Standard Channel 5/Value
//     PlcTask Inputs/GVL_iXlinker.EtherCAT_Master_EJxxxx.Beckhoff_EJ3xxx.A_0007_EJ3068_0000_0021.AI_Standard_Channel_6.Value <-> AI Standard Channel 6/Value
//     PlcTask Inputs/GVL_iXlinker.EtherCAT_Master_EJxxxx.Beckhoff_EJ3xxx.A_0007_EJ3068_0000_0021.AI_Standard_Channel_7.Value <-> AI Standard Channel 7/Value
//     PlcTask Inputs/GVL_iXlinker.EtherCAT_Master_EJxxxx.Beckhoff_EJ3xxx.A_0007_EJ3068_0000_0021.AI_Standard_Channel_8.Value <-> AI Standard Channel 8/Value
//     PlcTask Inputs/GVL_iXlinker.EtherCAT_Master_EJxxxx.Beckhoff_EJ3xxx.A_0007_EJ3068_0000_0021.WcState.WcState <-> WcState/WcState
//     PlcTask Inputs/GVL_iXlinker.EtherCAT_Master_EJxxxx.Beckhoff_EJ3xxx.A_0007_EJ3068_0000_0021.WcState.InputToggle <-> WcState/InputToggle
//     PlcTask Inputs/GVL_iXlinker.EtherCAT_Master_EJxxxx.Beckhoff_EJ3xxx.A_0007_EJ3068_0000_0021.InfoData.AdsAddr <-> InfoData/AdsAddr
//     PlcTask Inputs/GVL_iXlinker.EtherCAT_Master_EJxxxx.Beckhoff_EJ3xxx.A_0007_EJ3068_0000_0021.InfoData.State <-> InfoData/State
//   PLC/PLC Instance <-> EtherCAT Master EJxxxx/Beckhoff EJ3xxx/A_0008(EJ3104-0000-0019)
//     PlcTask Inputs/GVL_iXlinker.EtherCAT_Master_EJxxxx.Beckhoff_EJ3xxx.A_0008_EJ3104_0000_0019.AI_Standard_Channel_1.Status/Underrange <-> AI Standard Channel 1/Status/Underrange
//     PlcTask Inputs/GVL_iXlinker.EtherCAT_Master_EJxxxx.Beckhoff_EJ3xxx.A_0008_EJ3104_0000_0019.AI_Standard_Channel_2.Status/Underrange <-> AI Standard Channel 2/Status/Underrange
//     PlcTask Inputs/GVL_iXlinker.EtherCAT_Master_EJxxxx.Beckhoff_EJ3xxx.A_0008_EJ3104_0000_0019.AI_Standard_Channel_3.Status/Underrange <-> AI Standard Channel 3/Status/Underrange
//     PlcTask Inputs/GVL_iXlinker.EtherCAT_Master_EJxxxx.Beckhoff_EJ3xxx.A_0008_EJ3104_0000_0019.AI_Standard_Channel_4.Status/Underrange <-> AI Standard Channel 4/Status/Underrange
//     PlcTask Inputs/GVL_iXlinker.EtherCAT_Master_EJxxxx.Beckhoff_EJ3xxx.A_0008_EJ3104_0000_0019.AI_Standard_Channel_1.Status/Overrange <-> AI Standard Channel 1/Status/Overrange
//     PlcTask Inputs/GVL_iXlinker.EtherCAT_Master_EJxxxx.Beckhoff_EJ3xxx.A_0008_EJ3104_0000_0019.AI_Standard_Channel_2.Status/Overrange <-> AI Standard Channel 2/Status/Overrange
//     PlcTask Inputs/GVL_iXlinker.EtherCAT_Master_EJxxxx.Beckhoff_EJ3xxx.A_0008_EJ3104_0000_0019.AI_Standard_Channel_3.Status/Overrange <-> AI Standard Channel 3/Status/Overrange
//     PlcTask Inputs/GVL_iXlinker.EtherCAT_Master_EJxxxx.Beckhoff_EJ3xxx.A_0008_EJ3104_0000_0019.AI_Standard_Channel_4.Status/Overrange <-> AI Standard Channel 4/Status/Overrange
//     PlcTask Inputs/GVL_iXlinker.EtherCAT_Master_EJxxxx.Beckhoff_EJ3xxx.A_0008_EJ3104_0000_0019.AI_Standard_Channel_1.Status/Limit_1 <-> AI Standard Channel 1/Status/Limit 1
//     PlcTask Inputs/GVL_iXlinker.EtherCAT_Master_EJxxxx.Beckhoff_EJ3xxx.A_0008_EJ3104_0000_0019.AI_Standard_Channel_1.Status/Limit_2 <-> AI Standard Channel 1/Status/Limit 2
//     PlcTask Inputs/GVL_iXlinker.EtherCAT_Master_EJxxxx.Beckhoff_EJ3xxx.A_0008_EJ3104_0000_0019.AI_Standard_Channel_2.Status/Limit_1 <-> AI Standard Channel 2/Status/Limit 1
//     PlcTask Inputs/GVL_iXlinker.EtherCAT_Master_EJxxxx.Beckhoff_EJ3xxx.A_0008_EJ3104_0000_0019.AI_Standard_Channel_2.Status/Limit_2 <-> AI Standard Channel 2/Status/Limit 2
//     PlcTask Inputs/GVL_iXlinker.EtherCAT_Master_EJxxxx.Beckhoff_EJ3xxx.A_0008_EJ3104_0000_0019.AI_Standard_Channel_3.Status/Limit_1 <-> AI Standard Channel 3/Status/Limit 1
//     PlcTask Inputs/GVL_iXlinker.EtherCAT_Master_EJxxxx.Beckhoff_EJ3xxx.A_0008_EJ3104_0000_0019.AI_Standard_Channel_3.Status/Limit_2 <-> AI Standard Channel 3/Status/Limit 2
//     PlcTask Inputs/GVL_iXlinker.EtherCAT_Master_EJxxxx.Beckhoff_EJ3xxx.A_0008_EJ3104_0000_0019.AI_Standard_Channel_4.Status/Limit_1 <-> AI Standard Channel 4/Status/Limit 1
//     PlcTask Inputs/GVL_iXlinker.EtherCAT_Master_EJxxxx.Beckhoff_EJ3xxx.A_0008_EJ3104_0000_0019.AI_Standard_Channel_4.Status/Limit_2 <-> AI Standard Channel 4/Status/Limit 2
//     PlcTask Inputs/GVL_iXlinker.EtherCAT_Master_EJxxxx.Beckhoff_EJ3xxx.A_0008_EJ3104_0000_0019.AI_Standard_Channel_1.Status/Error <-> AI Standard Channel 1/Status/Error
//     PlcTask Inputs/GVL_iXlinker.EtherCAT_Master_EJxxxx.Beckhoff_EJ3xxx.A_0008_EJ3104_0000_0019.AI_Standard_Channel_2.Status/Error <-> AI Standard Channel 2/Status/Error
//     PlcTask Inputs/GVL_iXlinker.EtherCAT_Master_EJxxxx.Beckhoff_EJ3xxx.A_0008_EJ3104_0000_0019.AI_Standard_Channel_3.Status/Error <-> AI Standard Channel 3/Status/Error
//     PlcTask Inputs/GVL_iXlinker.EtherCAT_Master_EJxxxx.Beckhoff_EJ3xxx.A_0008_EJ3104_0000_0019.AI_Standard_Channel_4.Status/Error <-> AI Standard Channel 4/Status/Error
//     PlcTask Inputs/GVL_iXlinker.EtherCAT_Master_EJxxxx.Beckhoff_EJ3xxx.A_0008_EJ3104_0000_0019.AI_Standard_Channel_1.Status/Sync_error <-> AI Standard Channel 1/Status/Sync error
//     PlcTask Inputs/GVL_iXlinker.EtherCAT_Master_EJxxxx.Beckhoff_EJ3xxx.A_0008_EJ3104_0000_0019.AI_Standard_Channel_2.Status/Sync_error <-> AI Standard Channel 2/Status/Sync error
//     PlcTask Inputs/GVL_iXlinker.EtherCAT_Master_EJxxxx.Beckhoff_EJ3xxx.A_0008_EJ3104_0000_0019.AI_Standard_Channel_3.Status/Sync_error <-> AI Standard Channel 3/Status/Sync error
//     PlcTask Inputs/GVL_iXlinker.EtherCAT_Master_EJxxxx.Beckhoff_EJ3xxx.A_0008_EJ3104_0000_0019.AI_Standard_Channel_4.Status/Sync_error <-> AI Standard Channel 4/Status/Sync error
//     PlcTask Inputs/GVL_iXlinker.EtherCAT_Master_EJxxxx.Beckhoff_EJ3xxx.A_0008_EJ3104_0000_0019.AI_Standard_Channel_1.Status/TxPDO_State <-> AI Standard Channel 1/Status/TxPDO State
//     PlcTask Inputs/GVL_iXlinker.EtherCAT_Master_EJxxxx.Beckhoff_EJ3xxx.A_0008_EJ3104_0000_0019.AI_Standard_Channel_2.Status/TxPDO_State <-> AI Standard Channel 2/Status/TxPDO State
//     PlcTask Inputs/GVL_iXlinker.EtherCAT_Master_EJxxxx.Beckhoff_EJ3xxx.A_0008_EJ3104_0000_0019.AI_Standard_Channel_3.Status/TxPDO_State <-> AI Standard Channel 3/Status/TxPDO State
//     PlcTask Inputs/GVL_iXlinker.EtherCAT_Master_EJxxxx.Beckhoff_EJ3xxx.A_0008_EJ3104_0000_0019.AI_Standard_Channel_4.Status/TxPDO_State <-> AI Standard Channel 4/Status/TxPDO State
//     PlcTask Inputs/GVL_iXlinker.EtherCAT_Master_EJxxxx.Beckhoff_EJ3xxx.A_0008_EJ3104_0000_0019.AI_Standard_Channel_1.Status/TxPDO_Toggle <-> AI Standard Channel 1/Status/TxPDO Toggle
//     PlcTask Inputs/GVL_iXlinker.EtherCAT_Master_EJxxxx.Beckhoff_EJ3xxx.A_0008_EJ3104_0000_0019.AI_Standard_Channel_2.Status/TxPDO_Toggle <-> AI Standard Channel 2/Status/TxPDO Toggle
//     PlcTask Inputs/GVL_iXlinker.EtherCAT_Master_EJxxxx.Beckhoff_EJ3xxx.A_0008_EJ3104_0000_0019.AI_Standard_Channel_3.Status/TxPDO_Toggle <-> AI Standard Channel 3/Status/TxPDO Toggle
//     PlcTask Inputs/GVL_iXlinker.EtherCAT_Master_EJxxxx.Beckhoff_EJ3xxx.A_0008_EJ3104_0000_0019.AI_Standard_Channel_4.Status/TxPDO_Toggle <-> AI Standard Channel 4/Status/TxPDO Toggle
//     PlcTask Inputs/GVL_iXlinker.EtherCAT_Master_EJxxxx.Beckhoff_EJ3xxx.A_0008_EJ3104_0000_0019.AI_Standard_Channel_1.Value <-> AI Standard Channel 1/Value
//     PlcTask Inputs/GVL_iXlinker.EtherCAT_Master_EJxxxx.Beckhoff_EJ3xxx.A_0008_EJ3104_0000_0019.AI_Standard_Channel_2.Value <-> AI Standard Channel 2/Value
//     PlcTask Inputs/GVL_iXlinker.EtherCAT_Master_EJxxxx.Beckhoff_EJ3xxx.A_0008_EJ3104_0000_0019.AI_Standard_Channel_3.Value <-> AI Standard Channel 3/Value
//     PlcTask Inputs/GVL_iXlinker.EtherCAT_Master_EJxxxx.Beckhoff_EJ3xxx.A_0008_EJ3104_0000_0019.AI_Standard_Channel_4.Value <-> AI Standard Channel 4/Value
//     PlcTask Inputs/GVL_iXlinker.EtherCAT_Master_EJxxxx.Beckhoff_EJ3xxx.A_0008_EJ3104_0000_0019.WcState.WcState <-> WcState/WcState
//     PlcTask Inputs/GVL_iXlinker.EtherCAT_Master_EJxxxx.Beckhoff_EJ3xxx.A_0008_EJ3104_0000_0019.WcState.InputToggle <-> WcState/InputToggle
//     PlcTask Inputs/GVL_iXlinker.EtherCAT_Master_EJxxxx.Beckhoff_EJ3xxx.A_0008_EJ3104_0000_0019.InfoData.AdsAddr <-> InfoData/AdsAddr
//     PlcTask Inputs/GVL_iXlinker.EtherCAT_Master_EJxxxx.Beckhoff_EJ3xxx.A_0008_EJ3104_0000_0019.InfoData.State <-> InfoData/State
//   PLC/PLC Instance <-> EtherCAT Master EJxxxx/Beckhoff EJ3xxx/A_0009(EJ3104-0000-0020)
//     PlcTask Inputs/GVL_iXlinker.EtherCAT_Master_EJxxxx.Beckhoff_EJ3xxx.A_0009_EJ3104_0000_0020.AI_Standard_Channel_1.Status/Underrange <-> AI Standard Channel 1/Status/Underrange
//     PlcTask Inputs/GVL_iXlinker.EtherCAT_Master_EJxxxx.Beckhoff_EJ3xxx.A_0009_EJ3104_0000_0020.AI_Standard_Channel_2.Status/Underrange <-> AI Standard Channel 2/Status/Underrange
//     PlcTask Inputs/GVL_iXlinker.EtherCAT_Master_EJxxxx.Beckhoff_EJ3xxx.A_0009_EJ3104_0000_0020.AI_Standard_Channel_3.Status/Underrange <-> AI Standard Channel 3/Status/Underrange
//     PlcTask Inputs/GVL_iXlinker.EtherCAT_Master_EJxxxx.Beckhoff_EJ3xxx.A_0009_EJ3104_0000_0020.AI_Standard_Channel_4.Status/Underrange <-> AI Standard Channel 4/Status/Underrange
//     PlcTask Inputs/GVL_iXlinker.EtherCAT_Master_EJxxxx.Beckhoff_EJ3xxx.A_0009_EJ3104_0000_0020.AI_Standard_Channel_1.Status/Overrange <-> AI Standard Channel 1/Status/Overrange
//     PlcTask Inputs/GVL_iXlinker.EtherCAT_Master_EJxxxx.Beckhoff_EJ3xxx.A_0009_EJ3104_0000_0020.AI_Standard_Channel_2.Status/Overrange <-> AI Standard Channel 2/Status/Overrange
//     PlcTask Inputs/GVL_iXlinker.EtherCAT_Master_EJxxxx.Beckhoff_EJ3xxx.A_0009_EJ3104_0000_0020.AI_Standard_Channel_3.Status/Overrange <-> AI Standard Channel 3/Status/Overrange
//     PlcTask Inputs/GVL_iXlinker.EtherCAT_Master_EJxxxx.Beckhoff_EJ3xxx.A_0009_EJ3104_0000_0020.AI_Standard_Channel_4.Status/Overrange <-> AI Standard Channel 4/Status/Overrange
//     PlcTask Inputs/GVL_iXlinker.EtherCAT_Master_EJxxxx.Beckhoff_EJ3xxx.A_0009_EJ3104_0000_0020.AI_Standard_Channel_1.Status/Limit_1 <-> AI Standard Channel 1/Status/Limit 1
//     PlcTask Inputs/GVL_iXlinker.EtherCAT_Master_EJxxxx.Beckhoff_EJ3xxx.A_0009_EJ3104_0000_0020.AI_Standard_Channel_1.Status/Limit_2 <-> AI Standard Channel 1/Status/Limit 2
//     PlcTask Inputs/GVL_iXlinker.EtherCAT_Master_EJxxxx.Beckhoff_EJ3xxx.A_0009_EJ3104_0000_0020.AI_Standard_Channel_2.Status/Limit_1 <-> AI Standard Channel 2/Status/Limit 1
//     PlcTask Inputs/GVL_iXlinker.EtherCAT_Master_EJxxxx.Beckhoff_EJ3xxx.A_0009_EJ3104_0000_0020.AI_Standard_Channel_2.Status/Limit_2 <-> AI Standard Channel 2/Status/Limit 2
//     PlcTask Inputs/GVL_iXlinker.EtherCAT_Master_EJxxxx.Beckhoff_EJ3xxx.A_0009_EJ3104_0000_0020.AI_Standard_Channel_3.Status/Limit_1 <-> AI Standard Channel 3/Status/Limit 1
//     PlcTask Inputs/GVL_iXlinker.EtherCAT_Master_EJxxxx.Beckhoff_EJ3xxx.A_0009_EJ3104_0000_0020.AI_Standard_Channel_3.Status/Limit_2 <-> AI Standard Channel 3/Status/Limit 2
//     PlcTask Inputs/GVL_iXlinker.EtherCAT_Master_EJxxxx.Beckhoff_EJ3xxx.A_0009_EJ3104_0000_0020.AI_Standard_Channel_4.Status/Limit_1 <-> AI Standard Channel 4/Status/Limit 1
//     PlcTask Inputs/GVL_iXlinker.EtherCAT_Master_EJxxxx.Beckhoff_EJ3xxx.A_0009_EJ3104_0000_0020.AI_Standard_Channel_4.Status/Limit_2 <-> AI Standard Channel 4/Status/Limit 2
//     PlcTask Inputs/GVL_iXlinker.EtherCAT_Master_EJxxxx.Beckhoff_EJ3xxx.A_0009_EJ3104_0000_0020.AI_Standard_Channel_1.Status/Error <-> AI Standard Channel 1/Status/Error
//     PlcTask Inputs/GVL_iXlinker.EtherCAT_Master_EJxxxx.Beckhoff_EJ3xxx.A_0009_EJ3104_0000_0020.AI_Standard_Channel_2.Status/Error <-> AI Standard Channel 2/Status/Error
//     PlcTask Inputs/GVL_iXlinker.EtherCAT_Master_EJxxxx.Beckhoff_EJ3xxx.A_0009_EJ3104_0000_0020.AI_Standard_Channel_3.Status/Error <-> AI Standard Channel 3/Status/Error
//     PlcTask Inputs/GVL_iXlinker.EtherCAT_Master_EJxxxx.Beckhoff_EJ3xxx.A_0009_EJ3104_0000_0020.AI_Standard_Channel_4.Status/Error <-> AI Standard Channel 4/Status/Error
//     PlcTask Inputs/GVL_iXlinker.EtherCAT_Master_EJxxxx.Beckhoff_EJ3xxx.A_0009_EJ3104_0000_0020.AI_Standard_Channel_1.Status/Sync_error <-> AI Standard Channel 1/Status/Sync error
//     PlcTask Inputs/GVL_iXlinker.EtherCAT_Master_EJxxxx.Beckhoff_EJ3xxx.A_0009_EJ3104_0000_0020.AI_Standard_Channel_2.Status/Sync_error <-> AI Standard Channel 2/Status/Sync error
//     PlcTask Inputs/GVL_iXlinker.EtherCAT_Master_EJxxxx.Beckhoff_EJ3xxx.A_0009_EJ3104_0000_0020.AI_Standard_Channel_3.Status/Sync_error <-> AI Standard Channel 3/Status/Sync error
//     PlcTask Inputs/GVL_iXlinker.EtherCAT_Master_EJxxxx.Beckhoff_EJ3xxx.A_0009_EJ3104_0000_0020.AI_Standard_Channel_4.Status/Sync_error <-> AI Standard Channel 4/Status/Sync error
//     PlcTask Inputs/GVL_iXlinker.EtherCAT_Master_EJxxxx.Beckhoff_EJ3xxx.A_0009_EJ3104_0000_0020.AI_Standard_Channel_1.Status/TxPDO_State <-> AI Standard Channel 1/Status/TxPDO State
//     PlcTask Inputs/GVL_iXlinker.EtherCAT_Master_EJxxxx.Beckhoff_EJ3xxx.A_0009_EJ3104_0000_0020.AI_Standard_Channel_2.Status/TxPDO_State <-> AI Standard Channel 2/Status/TxPDO State
//     PlcTask Inputs/GVL_iXlinker.EtherCAT_Master_EJxxxx.Beckhoff_EJ3xxx.A_0009_EJ3104_0000_0020.AI_Standard_Channel_3.Status/TxPDO_State <-> AI Standard Channel 3/Status/TxPDO State
//     PlcTask Inputs/GVL_iXlinker.EtherCAT_Master_EJxxxx.Beckhoff_EJ3xxx.A_0009_EJ3104_0000_0020.AI_Standard_Channel_4.Status/TxPDO_State <-> AI Standard Channel 4/Status/TxPDO State
//     PlcTask Inputs/GVL_iXlinker.EtherCAT_Master_EJxxxx.Beckhoff_EJ3xxx.A_0009_EJ3104_0000_0020.AI_Standard_Channel_1.Status/TxPDO_Toggle <-> AI Standard Channel 1/Status/TxPDO Toggle
//     PlcTask Inputs/GVL_iXlinker.EtherCAT_Master_EJxxxx.Beckhoff_EJ3xxx.A_0009_EJ3104_0000_0020.AI_Standard_Channel_2.Status/TxPDO_Toggle <-> AI Standard Channel 2/Status/TxPDO Toggle
//     PlcTask Inputs/GVL_iXlinker.EtherCAT_Master_EJxxxx.Beckhoff_EJ3xxx.A_0009_EJ3104_0000_0020.AI_Standard_Channel_3.Status/TxPDO_Toggle <-> AI Standard Channel 3/Status/TxPDO Toggle
//     PlcTask Inputs/GVL_iXlinker.EtherCAT_Master_EJxxxx.Beckhoff_EJ3xxx.A_0009_EJ3104_0000_0020.AI_Standard_Channel_4.Status/TxPDO_Toggle <-> AI Standard Channel 4/Status/TxPDO Toggle
//     PlcTask Inputs/GVL_iXlinker.EtherCAT_Master_EJxxxx.Beckhoff_EJ3xxx.A_0009_EJ3104_0000_0020.AI_Standard_Channel_1.Value <-> AI Standard Channel 1/Value
//     PlcTask Inputs/GVL_iXlinker.EtherCAT_Master_EJxxxx.Beckhoff_EJ3xxx.A_0009_EJ3104_0000_0020.AI_Standard_Channel_2.Value <-> AI Standard Channel 2/Value
//     PlcTask Inputs/GVL_iXlinker.EtherCAT_Master_EJxxxx.Beckhoff_EJ3xxx.A_0009_EJ3104_0000_0020.AI_Standard_Channel_3.Value <-> AI Standard Channel 3/Value
//     PlcTask Inputs/GVL_iXlinker.EtherCAT_Master_EJxxxx.Beckhoff_EJ3xxx.A_0009_EJ3104_0000_0020.AI_Standard_Channel_4.Value <-> AI Standard Channel 4/Value
//     PlcTask Inputs/GVL_iXlinker.EtherCAT_Master_EJxxxx.Beckhoff_EJ3xxx.A_0009_EJ3104_0000_0020.WcState.WcState <-> WcState/WcState
//     PlcTask Inputs/GVL_iXlinker.EtherCAT_Master_EJxxxx.Beckhoff_EJ3xxx.A_0009_EJ3104_0000_0020.WcState.InputToggle <-> WcState/InputToggle
//     PlcTask Inputs/GVL_iXlinker.EtherCAT_Master_EJxxxx.Beckhoff_EJ3xxx.A_0009_EJ3104_0000_0020.InfoData.AdsAddr <-> InfoData/AdsAddr
//     PlcTask Inputs/GVL_iXlinker.EtherCAT_Master_EJxxxx.Beckhoff_EJ3xxx.A_0009_EJ3104_0000_0020.InfoData.State <-> InfoData/State
//   PLC/PLC Instance <-> EtherCAT Master EJxxxx/Beckhoff EJ3xxx/A_0010(EJ3104-0000-0021)
//     PlcTask Inputs/GVL_iXlinker.EtherCAT_Master_EJxxxx.Beckhoff_EJ3xxx.A_0010_EJ3104_0000_0021.AI_Standard_Channel_1.Status/Underrange <-> AI Standard Channel 1/Status/Underrange
//     PlcTask Inputs/GVL_iXlinker.EtherCAT_Master_EJxxxx.Beckhoff_EJ3xxx.A_0010_EJ3104_0000_0021.AI_Standard_Channel_2.Status/Underrange <-> AI Standard Channel 2/Status/Underrange
//     PlcTask Inputs/GVL_iXlinker.EtherCAT_Master_EJxxxx.Beckhoff_EJ3xxx.A_0010_EJ3104_0000_0021.AI_Standard_Channel_3.Status/Underrange <-> AI Standard Channel 3/Status/Underrange
//     PlcTask Inputs/GVL_iXlinker.EtherCAT_Master_EJxxxx.Beckhoff_EJ3xxx.A_0010_EJ3104_0000_0021.AI_Standard_Channel_4.Status/Underrange <-> AI Standard Channel 4/Status/Underrange
//     PlcTask Inputs/GVL_iXlinker.EtherCAT_Master_EJxxxx.Beckhoff_EJ3xxx.A_0010_EJ3104_0000_0021.AI_Standard_Channel_1.Status/Overrange <-> AI Standard Channel 1/Status/Overrange
//     PlcTask Inputs/GVL_iXlinker.EtherCAT_Master_EJxxxx.Beckhoff_EJ3xxx.A_0010_EJ3104_0000_0021.AI_Standard_Channel_2.Status/Overrange <-> AI Standard Channel 2/Status/Overrange
//     PlcTask Inputs/GVL_iXlinker.EtherCAT_Master_EJxxxx.Beckhoff_EJ3xxx.A_0010_EJ3104_0000_0021.AI_Standard_Channel_3.Status/Overrange <-> AI Standard Channel 3/Status/Overrange
//     PlcTask Inputs/GVL_iXlinker.EtherCAT_Master_EJxxxx.Beckhoff_EJ3xxx.A_0010_EJ3104_0000_0021.AI_Standard_Channel_4.Status/Overrange <-> AI Standard Channel 4/Status/Overrange
//     PlcTask Inputs/GVL_iXlinker.EtherCAT_Master_EJxxxx.Beckhoff_EJ3xxx.A_0010_EJ3104_0000_0021.AI_Standard_Channel_1.Status/Limit_1 <-> AI Standard Channel 1/Status/Limit 1
//     PlcTask Inputs/GVL_iXlinker.EtherCAT_Master_EJxxxx.Beckhoff_EJ3xxx.A_0010_EJ3104_0000_0021.AI_Standard_Channel_1.Status/Limit_2 <-> AI Standard Channel 1/Status/Limit 2
//     PlcTask Inputs/GVL_iXlinker.EtherCAT_Master_EJxxxx.Beckhoff_EJ3xxx.A_0010_EJ3104_0000_0021.AI_Standard_Channel_2.Status/Limit_1 <-> AI Standard Channel 2/Status/Limit 1
//     PlcTask Inputs/GVL_iXlinker.EtherCAT_Master_EJxxxx.Beckhoff_EJ3xxx.A_0010_EJ3104_0000_0021.AI_Standard_Channel_2.Status/Limit_2 <-> AI Standard Channel 2/Status/Limit 2
//     PlcTask Inputs/GVL_iXlinker.EtherCAT_Master_EJxxxx.Beckhoff_EJ3xxx.A_0010_EJ3104_0000_0021.AI_Standard_Channel_3.Status/Limit_1 <-> AI Standard Channel 3/Status/Limit 1
//     PlcTask Inputs/GVL_iXlinker.EtherCAT_Master_EJxxxx.Beckhoff_EJ3xxx.A_0010_EJ3104_0000_0021.AI_Standard_Channel_3.Status/Limit_2 <-> AI Standard Channel 3/Status/Limit 2
//     PlcTask Inputs/GVL_iXlinker.EtherCAT_Master_EJxxxx.Beckhoff_EJ3xxx.A_0010_EJ3104_0000_0021.AI_Standard_Channel_4.Status/Limit_1 <-> AI Standard Channel 4/Status/Limit 1
//     PlcTask Inputs/GVL_iXlinker.EtherCAT_Master_EJxxxx.Beckhoff_EJ3xxx.A_0010_EJ3104_0000_0021.AI_Standard_Channel_4.Status/Limit_2 <-> AI Standard Channel 4/Status/Limit 2
//     PlcTask Inputs/GVL_iXlinker.EtherCAT_Master_EJxxxx.Beckhoff_EJ3xxx.A_0010_EJ3104_0000_0021.AI_Standard_Channel_1.Status/Error <-> AI Standard Channel 1/Status/Error
//     PlcTask Inputs/GVL_iXlinker.EtherCAT_Master_EJxxxx.Beckhoff_EJ3xxx.A_0010_EJ3104_0000_0021.AI_Standard_Channel_2.Status/Error <-> AI Standard Channel 2/Status/Error
//     PlcTask Inputs/GVL_iXlinker.EtherCAT_Master_EJxxxx.Beckhoff_EJ3xxx.A_0010_EJ3104_0000_0021.AI_Standard_Channel_3.Status/Error <-> AI Standard Channel 3/Status/Error
//     PlcTask Inputs/GVL_iXlinker.EtherCAT_Master_EJxxxx.Beckhoff_EJ3xxx.A_0010_EJ3104_0000_0021.AI_Standard_Channel_4.Status/Error <-> AI Standard Channel 4/Status/Error
//     PlcTask Inputs/GVL_iXlinker.EtherCAT_Master_EJxxxx.Beckhoff_EJ3xxx.A_0010_EJ3104_0000_0021.AI_Standard_Channel_1.Status/Sync_error <-> AI Standard Channel 1/Status/Sync error
//     PlcTask Inputs/GVL_iXlinker.EtherCAT_Master_EJxxxx.Beckhoff_EJ3xxx.A_0010_EJ3104_0000_0021.AI_Standard_Channel_2.Status/Sync_error <-> AI Standard Channel 2/Status/Sync error
//     PlcTask Inputs/GVL_iXlinker.EtherCAT_Master_EJxxxx.Beckhoff_EJ3xxx.A_0010_EJ3104_0000_0021.AI_Standard_Channel_3.Status/Sync_error <-> AI Standard Channel 3/Status/Sync error
//     PlcTask Inputs/GVL_iXlinker.EtherCAT_Master_EJxxxx.Beckhoff_EJ3xxx.A_0010_EJ3104_0000_0021.AI_Standard_Channel_4.Status/Sync_error <-> AI Standard Channel 4/Status/Sync error
//     PlcTask Inputs/GVL_iXlinker.EtherCAT_Master_EJxxxx.Beckhoff_EJ3xxx.A_0010_EJ3104_0000_0021.AI_Standard_Channel_1.Status/TxPDO_State <-> AI Standard Channel 1/Status/TxPDO State
//     PlcTask Inputs/GVL_iXlinker.EtherCAT_Master_EJxxxx.Beckhoff_EJ3xxx.A_0010_EJ3104_0000_0021.AI_Standard_Channel_2.Status/TxPDO_State <-> AI Standard Channel 2/Status/TxPDO State
//     PlcTask Inputs/GVL_iXlinker.EtherCAT_Master_EJxxxx.Beckhoff_EJ3xxx.A_0010_EJ3104_0000_0021.AI_Standard_Channel_3.Status/TxPDO_State <-> AI Standard Channel 3/Status/TxPDO State
//     PlcTask Inputs/GVL_iXlinker.EtherCAT_Master_EJxxxx.Beckhoff_EJ3xxx.A_0010_EJ3104_0000_0021.AI_Standard_Channel_4.Status/TxPDO_State <-> AI Standard Channel 4/Status/TxPDO State
//     PlcTask Inputs/GVL_iXlinker.EtherCAT_Master_EJxxxx.Beckhoff_EJ3xxx.A_0010_EJ3104_0000_0021.AI_Standard_Channel_1.Status/TxPDO_Toggle <-> AI Standard Channel 1/Status/TxPDO Toggle
//     PlcTask Inputs/GVL_iXlinker.EtherCAT_Master_EJxxxx.Beckhoff_EJ3xxx.A_0010_EJ3104_0000_0021.AI_Standard_Channel_2.Status/TxPDO_Toggle <-> AI Standard Channel 2/Status/TxPDO Toggle
//     PlcTask Inputs/GVL_iXlinker.EtherCAT_Master_EJxxxx.Beckhoff_EJ3xxx.A_0010_EJ3104_0000_0021.AI_Standard_Channel_3.Status/TxPDO_Toggle <-> AI Standard Channel 3/Status/TxPDO Toggle
//     PlcTask Inputs/GVL_iXlinker.EtherCAT_Master_EJxxxx.Beckhoff_EJ3xxx.A_0010_EJ3104_0000_0021.AI_Standard_Channel_4.Status/TxPDO_Toggle <-> AI Standard Channel 4/Status/TxPDO Toggle
//     PlcTask Inputs/GVL_iXlinker.EtherCAT_Master_EJxxxx.Beckhoff_EJ3xxx.A_0010_EJ3104_0000_0021.AI_Standard_Channel_1.Value <-> AI Standard Channel 1/Value
//     PlcTask Inputs/GVL_iXlinker.EtherCAT_Master_EJxxxx.Beckhoff_EJ3xxx.A_0010_EJ3104_0000_0021.AI_Standard_Channel_2.Value <-> AI Standard Channel 2/Value
//     PlcTask Inputs/GVL_iXlinker.EtherCAT_Master_EJxxxx.Beckhoff_EJ3xxx.A_0010_EJ3104_0000_0021.AI_Standard_Channel_3.Value <-> AI Standard Channel 3/Value
//     PlcTask Inputs/GVL_iXlinker.EtherCAT_Master_EJxxxx.Beckhoff_EJ3xxx.A_0010_EJ3104_0000_0021.AI_Standard_Channel_4.Value <-> AI Standard Channel 4/Value
//     PlcTask Inputs/GVL_iXlinker.EtherCAT_Master_EJxxxx.Beckhoff_EJ3xxx.A_0010_EJ3104_0000_0021.WcState.WcState <-> WcState/WcState
//     PlcTask Inputs/GVL_iXlinker.EtherCAT_Master_EJxxxx.Beckhoff_EJ3xxx.A_0010_EJ3104_0000_0021.WcState.InputToggle <-> WcState/InputToggle
//     PlcTask Inputs/GVL_iXlinker.EtherCAT_Master_EJxxxx.Beckhoff_EJ3xxx.A_0010_EJ3104_0000_0021.InfoData.AdsAddr <-> InfoData/AdsAddr
//     PlcTask Inputs/GVL_iXlinker.EtherCAT_Master_EJxxxx.Beckhoff_EJ3xxx.A_0010_EJ3104_0000_0021.InfoData.State <-> InfoData/State
//   PLC/PLC Instance <-> EtherCAT Master EJxxxx/Beckhoff EJ3xxx/A_0011(EJ3108-0000-0017)
//     PlcTask Inputs/GVL_iXlinker.EtherCAT_Master_EJxxxx.Beckhoff_EJ3xxx.A_0011_EJ3108_0000_0017.AI_Standard_Channel_1.Status/Underrange <-> AI Standard Channel 1/Status/Underrange
//     PlcTask Inputs/GVL_iXlinker.EtherCAT_Master_EJxxxx.Beckhoff_EJ3xxx.A_0011_EJ3108_0000_0017.AI_Standard_Channel_2.Status/Underrange <-> AI Standard Channel 2/Status/Underrange
//     PlcTask Inputs/GVL_iXlinker.EtherCAT_Master_EJxxxx.Beckhoff_EJ3xxx.A_0011_EJ3108_0000_0017.AI_Standard_Channel_3.Status/Underrange <-> AI Standard Channel 3/Status/Underrange
//     PlcTask Inputs/GVL_iXlinker.EtherCAT_Master_EJxxxx.Beckhoff_EJ3xxx.A_0011_EJ3108_0000_0017.AI_Standard_Channel_4.Status/Underrange <-> AI Standard Channel 4/Status/Underrange
//     PlcTask Inputs/GVL_iXlinker.EtherCAT_Master_EJxxxx.Beckhoff_EJ3xxx.A_0011_EJ3108_0000_0017.AI_Standard_Channel_5.Status/Underrange <-> AI Standard Channel 5/Status/Underrange
//     PlcTask Inputs/GVL_iXlinker.EtherCAT_Master_EJxxxx.Beckhoff_EJ3xxx.A_0011_EJ3108_0000_0017.AI_Standard_Channel_6.Status/Underrange <-> AI Standard Channel 6/Status/Underrange
//     PlcTask Inputs/GVL_iXlinker.EtherCAT_Master_EJxxxx.Beckhoff_EJ3xxx.A_0011_EJ3108_0000_0017.AI_Standard_Channel_7.Status/Underrange <-> AI Standard Channel 7/Status/Underrange
//     PlcTask Inputs/GVL_iXlinker.EtherCAT_Master_EJxxxx.Beckhoff_EJ3xxx.A_0011_EJ3108_0000_0017.AI_Standard_Channel_8.Status/Underrange <-> AI Standard Channel 8/Status/Underrange
//     PlcTask Inputs/GVL_iXlinker.EtherCAT_Master_EJxxxx.Beckhoff_EJ3xxx.A_0011_EJ3108_0000_0017.AI_Standard_Channel_1.Status/Overrange <-> AI Standard Channel 1/Status/Overrange
//     PlcTask Inputs/GVL_iXlinker.EtherCAT_Master_EJxxxx.Beckhoff_EJ3xxx.A_0011_EJ3108_0000_0017.AI_Standard_Channel_2.Status/Overrange <-> AI Standard Channel 2/Status/Overrange
//     PlcTask Inputs/GVL_iXlinker.EtherCAT_Master_EJxxxx.Beckhoff_EJ3xxx.A_0011_EJ3108_0000_0017.AI_Standard_Channel_3.Status/Overrange <-> AI Standard Channel 3/Status/Overrange
//     PlcTask Inputs/GVL_iXlinker.EtherCAT_Master_EJxxxx.Beckhoff_EJ3xxx.A_0011_EJ3108_0000_0017.AI_Standard_Channel_4.Status/Overrange <-> AI Standard Channel 4/Status/Overrange
//     PlcTask Inputs/GVL_iXlinker.EtherCAT_Master_EJxxxx.Beckhoff_EJ3xxx.A_0011_EJ3108_0000_0017.AI_Standard_Channel_5.Status/Overrange <-> AI Standard Channel 5/Status/Overrange
//     PlcTask Inputs/GVL_iXlinker.EtherCAT_Master_EJxxxx.Beckhoff_EJ3xxx.A_0011_EJ3108_0000_0017.AI_Standard_Channel_6.Status/Overrange <-> AI Standard Channel 6/Status/Overrange
//     PlcTask Inputs/GVL_iXlinker.EtherCAT_Master_EJxxxx.Beckhoff_EJ3xxx.A_0011_EJ3108_0000_0017.AI_Standard_Channel_7.Status/Overrange <-> AI Standard Channel 7/Status/Overrange
//     PlcTask Inputs/GVL_iXlinker.EtherCAT_Master_EJxxxx.Beckhoff_EJ3xxx.A_0011_EJ3108_0000_0017.AI_Standard_Channel_8.Status/Overrange <-> AI Standard Channel 8/Status/Overrange
//     PlcTask Inputs/GVL_iXlinker.EtherCAT_Master_EJxxxx.Beckhoff_EJ3xxx.A_0011_EJ3108_0000_0017.AI_Standard_Channel_1.Status/Limit_1 <-> AI Standard Channel 1/Status/Limit 1
//     PlcTask Inputs/GVL_iXlinker.EtherCAT_Master_EJxxxx.Beckhoff_EJ3xxx.A_0011_EJ3108_0000_0017.AI_Standard_Channel_1.Status/Limit_2 <-> AI Standard Channel 1/Status/Limit 2
//     PlcTask Inputs/GVL_iXlinker.EtherCAT_Master_EJxxxx.Beckhoff_EJ3xxx.A_0011_EJ3108_0000_0017.AI_Standard_Channel_2.Status/Limit_1 <-> AI Standard Channel 2/Status/Limit 1
//     PlcTask Inputs/GVL_iXlinker.EtherCAT_Master_EJxxxx.Beckhoff_EJ3xxx.A_0011_EJ3108_0000_0017.AI_Standard_Channel_2.Status/Limit_2 <-> AI Standard Channel 2/Status/Limit 2
//     PlcTask Inputs/GVL_iXlinker.EtherCAT_Master_EJxxxx.Beckhoff_EJ3xxx.A_0011_EJ3108_0000_0017.AI_Standard_Channel_3.Status/Limit_1 <-> AI Standard Channel 3/Status/Limit 1
//     PlcTask Inputs/GVL_iXlinker.EtherCAT_Master_EJxxxx.Beckhoff_EJ3xxx.A_0011_EJ3108_0000_0017.AI_Standard_Channel_3.Status/Limit_2 <-> AI Standard Channel 3/Status/Limit 2
//     PlcTask Inputs/GVL_iXlinker.EtherCAT_Master_EJxxxx.Beckhoff_EJ3xxx.A_0011_EJ3108_0000_0017.AI_Standard_Channel_4.Status/Limit_1 <-> AI Standard Channel 4/Status/Limit 1
//     PlcTask Inputs/GVL_iXlinker.EtherCAT_Master_EJxxxx.Beckhoff_EJ3xxx.A_0011_EJ3108_0000_0017.AI_Standard_Channel_4.Status/Limit_2 <-> AI Standard Channel 4/Status/Limit 2
//     PlcTask Inputs/GVL_iXlinker.EtherCAT_Master_EJxxxx.Beckhoff_EJ3xxx.A_0011_EJ3108_0000_0017.AI_Standard_Channel_5.Status/Limit_1 <-> AI Standard Channel 5/Status/Limit 1
//     PlcTask Inputs/GVL_iXlinker.EtherCAT_Master_EJxxxx.Beckhoff_EJ3xxx.A_0011_EJ3108_0000_0017.AI_Standard_Channel_5.Status/Limit_2 <-> AI Standard Channel 5/Status/Limit 2
//     PlcTask Inputs/GVL_iXlinker.EtherCAT_Master_EJxxxx.Beckhoff_EJ3xxx.A_0011_EJ3108_0000_0017.AI_Standard_Channel_6.Status/Limit_1 <-> AI Standard Channel 6/Status/Limit 1
//     PlcTask Inputs/GVL_iXlinker.EtherCAT_Master_EJxxxx.Beckhoff_EJ3xxx.A_0011_EJ3108_0000_0017.AI_Standard_Channel_6.Status/Limit_2 <-> AI Standard Channel 6/Status/Limit 2
//     PlcTask Inputs/GVL_iXlinker.EtherCAT_Master_EJxxxx.Beckhoff_EJ3xxx.A_0011_EJ3108_0000_0017.AI_Standard_Channel_7.Status/Limit_1 <-> AI Standard Channel 7/Status/Limit 1
//     PlcTask Inputs/GVL_iXlinker.EtherCAT_Master_EJxxxx.Beckhoff_EJ3xxx.A_0011_EJ3108_0000_0017.AI_Standard_Channel_7.Status/Limit_2 <-> AI Standard Channel 7/Status/Limit 2
//     PlcTask Inputs/GVL_iXlinker.EtherCAT_Master_EJxxxx.Beckhoff_EJ3xxx.A_0011_EJ3108_0000_0017.AI_Standard_Channel_8.Status/Limit_1 <-> AI Standard Channel 8/Status/Limit 1
//     PlcTask Inputs/GVL_iXlinker.EtherCAT_Master_EJxxxx.Beckhoff_EJ3xxx.A_0011_EJ3108_0000_0017.AI_Standard_Channel_8.Status/Limit_2 <-> AI Standard Channel 8/Status/Limit 2
//     PlcTask Inputs/GVL_iXlinker.EtherCAT_Master_EJxxxx.Beckhoff_EJ3xxx.A_0011_EJ3108_0000_0017.AI_Standard_Channel_1.Status/Error <-> AI Standard Channel 1/Status/Error
//     PlcTask Inputs/GVL_iXlinker.EtherCAT_Master_EJxxxx.Beckhoff_EJ3xxx.A_0011_EJ3108_0000_0017.AI_Standard_Channel_2.Status/Error <-> AI Standard Channel 2/Status/Error
//     PlcTask Inputs/GVL_iXlinker.EtherCAT_Master_EJxxxx.Beckhoff_EJ3xxx.A_0011_EJ3108_0000_0017.AI_Standard_Channel_3.Status/Error <-> AI Standard Channel 3/Status/Error
//     PlcTask Inputs/GVL_iXlinker.EtherCAT_Master_EJxxxx.Beckhoff_EJ3xxx.A_0011_EJ3108_0000_0017.AI_Standard_Channel_4.Status/Error <-> AI Standard Channel 4/Status/Error
//     PlcTask Inputs/GVL_iXlinker.EtherCAT_Master_EJxxxx.Beckhoff_EJ3xxx.A_0011_EJ3108_0000_0017.AI_Standard_Channel_5.Status/Error <-> AI Standard Channel 5/Status/Error
//     PlcTask Inputs/GVL_iXlinker.EtherCAT_Master_EJxxxx.Beckhoff_EJ3xxx.A_0011_EJ3108_0000_0017.AI_Standard_Channel_6.Status/Error <-> AI Standard Channel 6/Status/Error
//     PlcTask Inputs/GVL_iXlinker.EtherCAT_Master_EJxxxx.Beckhoff_EJ3xxx.A_0011_EJ3108_0000_0017.AI_Standard_Channel_7.Status/Error <-> AI Standard Channel 7/Status/Error
//     PlcTask Inputs/GVL_iXlinker.EtherCAT_Master_EJxxxx.Beckhoff_EJ3xxx.A_0011_EJ3108_0000_0017.AI_Standard_Channel_8.Status/Error <-> AI Standard Channel 8/Status/Error
//     PlcTask Inputs/GVL_iXlinker.EtherCAT_Master_EJxxxx.Beckhoff_EJ3xxx.A_0011_EJ3108_0000_0017.AI_Standard_Channel_1.Status/TxPDO_State <-> AI Standard Channel 1/Status/TxPDO State
//     PlcTask Inputs/GVL_iXlinker.EtherCAT_Master_EJxxxx.Beckhoff_EJ3xxx.A_0011_EJ3108_0000_0017.AI_Standard_Channel_2.Status/TxPDO_State <-> AI Standard Channel 2/Status/TxPDO State
//     PlcTask Inputs/GVL_iXlinker.EtherCAT_Master_EJxxxx.Beckhoff_EJ3xxx.A_0011_EJ3108_0000_0017.AI_Standard_Channel_3.Status/TxPDO_State <-> AI Standard Channel 3/Status/TxPDO State
//     PlcTask Inputs/GVL_iXlinker.EtherCAT_Master_EJxxxx.Beckhoff_EJ3xxx.A_0011_EJ3108_0000_0017.AI_Standard_Channel_4.Status/TxPDO_State <-> AI Standard Channel 4/Status/TxPDO State
//     PlcTask Inputs/GVL_iXlinker.EtherCAT_Master_EJxxxx.Beckhoff_EJ3xxx.A_0011_EJ3108_0000_0017.AI_Standard_Channel_5.Status/TxPDO_State <-> AI Standard Channel 5/Status/TxPDO State
//     PlcTask Inputs/GVL_iXlinker.EtherCAT_Master_EJxxxx.Beckhoff_EJ3xxx.A_0011_EJ3108_0000_0017.AI_Standard_Channel_6.Status/TxPDO_State <-> AI Standard Channel 6/Status/TxPDO State
//     PlcTask Inputs/GVL_iXlinker.EtherCAT_Master_EJxxxx.Beckhoff_EJ3xxx.A_0011_EJ3108_0000_0017.AI_Standard_Channel_7.Status/TxPDO_State <-> AI Standard Channel 7/Status/TxPDO State
//     PlcTask Inputs/GVL_iXlinker.EtherCAT_Master_EJxxxx.Beckhoff_EJ3xxx.A_0011_EJ3108_0000_0017.AI_Standard_Channel_8.Status/TxPDO_State <-> AI Standard Channel 8/Status/TxPDO State
//     PlcTask Inputs/GVL_iXlinker.EtherCAT_Master_EJxxxx.Beckhoff_EJ3xxx.A_0011_EJ3108_0000_0017.AI_Standard_Channel_1.Status/TxPDO_Toggle <-> AI Standard Channel 1/Status/TxPDO Toggle
//     PlcTask Inputs/GVL_iXlinker.EtherCAT_Master_EJxxxx.Beckhoff_EJ3xxx.A_0011_EJ3108_0000_0017.AI_Standard_Channel_2.Status/TxPDO_Toggle <-> AI Standard Channel 2/Status/TxPDO Toggle
//     PlcTask Inputs/GVL_iXlinker.EtherCAT_Master_EJxxxx.Beckhoff_EJ3xxx.A_0011_EJ3108_0000_0017.AI_Standard_Channel_3.Status/TxPDO_Toggle <-> AI Standard Channel 3/Status/TxPDO Toggle
//     PlcTask Inputs/GVL_iXlinker.EtherCAT_Master_EJxxxx.Beckhoff_EJ3xxx.A_0011_EJ3108_0000_0017.AI_Standard_Channel_4.Status/TxPDO_Toggle <-> AI Standard Channel 4/Status/TxPDO Toggle
//     PlcTask Inputs/GVL_iXlinker.EtherCAT_Master_EJxxxx.Beckhoff_EJ3xxx.A_0011_EJ3108_0000_0017.AI_Standard_Channel_5.Status/TxPDO_Toggle <-> AI Standard Channel 5/Status/TxPDO Toggle
//     PlcTask Inputs/GVL_iXlinker.EtherCAT_Master_EJxxxx.Beckhoff_EJ3xxx.A_0011_EJ3108_0000_0017.AI_Standard_Channel_6.Status/TxPDO_Toggle <-> AI Standard Channel 6/Status/TxPDO Toggle
//     PlcTask Inputs/GVL_iXlinker.EtherCAT_Master_EJxxxx.Beckhoff_EJ3xxx.A_0011_EJ3108_0000_0017.AI_Standard_Channel_7.Status/TxPDO_Toggle <-> AI Standard Channel 7/Status/TxPDO Toggle
//     PlcTask Inputs/GVL_iXlinker.EtherCAT_Master_EJxxxx.Beckhoff_EJ3xxx.A_0011_EJ3108_0000_0017.AI_Standard_Channel_8.Status/TxPDO_Toggle <-> AI Standard Channel 8/Status/TxPDO Toggle
//     PlcTask Inputs/GVL_iXlinker.EtherCAT_Master_EJxxxx.Beckhoff_EJ3xxx.A_0011_EJ3108_0000_0017.AI_Standard_Channel_1.Value <-> AI Standard Channel 1/Value
//     PlcTask Inputs/GVL_iXlinker.EtherCAT_Master_EJxxxx.Beckhoff_EJ3xxx.A_0011_EJ3108_0000_0017.AI_Standard_Channel_2.Value <-> AI Standard Channel 2/Value
//     PlcTask Inputs/GVL_iXlinker.EtherCAT_Master_EJxxxx.Beckhoff_EJ3xxx.A_0011_EJ3108_0000_0017.AI_Standard_Channel_3.Value <-> AI Standard Channel 3/Value
//     PlcTask Inputs/GVL_iXlinker.EtherCAT_Master_EJxxxx.Beckhoff_EJ3xxx.A_0011_EJ3108_0000_0017.AI_Standard_Channel_4.Value <-> AI Standard Channel 4/Value
//     PlcTask Inputs/GVL_iXlinker.EtherCAT_Master_EJxxxx.Beckhoff_EJ3xxx.A_0011_EJ3108_0000_0017.AI_Standard_Channel_5.Value <-> AI Standard Channel 5/Value
//     PlcTask Inputs/GVL_iXlinker.EtherCAT_Master_EJxxxx.Beckhoff_EJ3xxx.A_0011_EJ3108_0000_0017.AI_Standard_Channel_6.Value <-> AI Standard Channel 6/Value
//     PlcTask Inputs/GVL_iXlinker.EtherCAT_Master_EJxxxx.Beckhoff_EJ3xxx.A_0011_EJ3108_0000_0017.AI_Standard_Channel_7.Value <-> AI Standard Channel 7/Value
//     PlcTask Inputs/GVL_iXlinker.EtherCAT_Master_EJxxxx.Beckhoff_EJ3xxx.A_0011_EJ3108_0000_0017.AI_Standard_Channel_8.Value <-> AI Standard Channel 8/Value
//     PlcTask Inputs/GVL_iXlinker.EtherCAT_Master_EJxxxx.Beckhoff_EJ3xxx.A_0011_EJ3108_0000_0017.WcState.WcState <-> WcState/WcState
//     PlcTask Inputs/GVL_iXlinker.EtherCAT_Master_EJxxxx.Beckhoff_EJ3xxx.A_0011_EJ3108_0000_0017.WcState.InputToggle <-> WcState/InputToggle
//     PlcTask Inputs/GVL_iXlinker.EtherCAT_Master_EJxxxx.Beckhoff_EJ3xxx.A_0011_EJ3108_0000_0017.InfoData.AdsAddr <-> InfoData/AdsAddr
//     PlcTask Inputs/GVL_iXlinker.EtherCAT_Master_EJxxxx.Beckhoff_EJ3xxx.A_0011_EJ3108_0000_0017.InfoData.State <-> InfoData/State
//   PLC/PLC Instance <-> EtherCAT Master EJxxxx/Beckhoff EJ3xxx/A_0012(EJ3108-0000-0018)
//     PlcTask Inputs/GVL_iXlinker.EtherCAT_Master_EJxxxx.Beckhoff_EJ3xxx.A_0012_EJ3108_0000_0018.AI_Standard_Channel_1.Status/Underrange <-> AI Standard Channel 1/Status/Underrange
//     PlcTask Inputs/GVL_iXlinker.EtherCAT_Master_EJxxxx.Beckhoff_EJ3xxx.A_0012_EJ3108_0000_0018.AI_Standard_Channel_2.Status/Underrange <-> AI Standard Channel 2/Status/Underrange
//     PlcTask Inputs/GVL_iXlinker.EtherCAT_Master_EJxxxx.Beckhoff_EJ3xxx.A_0012_EJ3108_0000_0018.AI_Standard_Channel_3.Status/Underrange <-> AI Standard Channel 3/Status/Underrange
//     PlcTask Inputs/GVL_iXlinker.EtherCAT_Master_EJxxxx.Beckhoff_EJ3xxx.A_0012_EJ3108_0000_0018.AI_Standard_Channel_4.Status/Underrange <-> AI Standard Channel 4/Status/Underrange
//     PlcTask Inputs/GVL_iXlinker.EtherCAT_Master_EJxxxx.Beckhoff_EJ3xxx.A_0012_EJ3108_0000_0018.AI_Standard_Channel_5.Status/Underrange <-> AI Standard Channel 5/Status/Underrange
//     PlcTask Inputs/GVL_iXlinker.EtherCAT_Master_EJxxxx.Beckhoff_EJ3xxx.A_0012_EJ3108_0000_0018.AI_Standard_Channel_6.Status/Underrange <-> AI Standard Channel 6/Status/Underrange
//     PlcTask Inputs/GVL_iXlinker.EtherCAT_Master_EJxxxx.Beckhoff_EJ3xxx.A_0012_EJ3108_0000_0018.AI_Standard_Channel_7.Status/Underrange <-> AI Standard Channel 7/Status/Underrange
//     PlcTask Inputs/GVL_iXlinker.EtherCAT_Master_EJxxxx.Beckhoff_EJ3xxx.A_0012_EJ3108_0000_0018.AI_Standard_Channel_8.Status/Underrange <-> AI Standard Channel 8/Status/Underrange
//     PlcTask Inputs/GVL_iXlinker.EtherCAT_Master_EJxxxx.Beckhoff_EJ3xxx.A_0012_EJ3108_0000_0018.AI_Standard_Channel_1.Status/Overrange <-> AI Standard Channel 1/Status/Overrange
//     PlcTask Inputs/GVL_iXlinker.EtherCAT_Master_EJxxxx.Beckhoff_EJ3xxx.A_0012_EJ3108_0000_0018.AI_Standard_Channel_2.Status/Overrange <-> AI Standard Channel 2/Status/Overrange
//     PlcTask Inputs/GVL_iXlinker.EtherCAT_Master_EJxxxx.Beckhoff_EJ3xxx.A_0012_EJ3108_0000_0018.AI_Standard_Channel_3.Status/Overrange <-> AI Standard Channel 3/Status/Overrange
//     PlcTask Inputs/GVL_iXlinker.EtherCAT_Master_EJxxxx.Beckhoff_EJ3xxx.A_0012_EJ3108_0000_0018.AI_Standard_Channel_4.Status/Overrange <-> AI Standard Channel 4/Status/Overrange
//     PlcTask Inputs/GVL_iXlinker.EtherCAT_Master_EJxxxx.Beckhoff_EJ3xxx.A_0012_EJ3108_0000_0018.AI_Standard_Channel_5.Status/Overrange <-> AI Standard Channel 5/Status/Overrange
//     PlcTask Inputs/GVL_iXlinker.EtherCAT_Master_EJxxxx.Beckhoff_EJ3xxx.A_0012_EJ3108_0000_0018.AI_Standard_Channel_6.Status/Overrange <-> AI Standard Channel 6/Status/Overrange
//     PlcTask Inputs/GVL_iXlinker.EtherCAT_Master_EJxxxx.Beckhoff_EJ3xxx.A_0012_EJ3108_0000_0018.AI_Standard_Channel_7.Status/Overrange <-> AI Standard Channel 7/Status/Overrange
//     PlcTask Inputs/GVL_iXlinker.EtherCAT_Master_EJxxxx.Beckhoff_EJ3xxx.A_0012_EJ3108_0000_0018.AI_Standard_Channel_8.Status/Overrange <-> AI Standard Channel 8/Status/Overrange
//     PlcTask Inputs/GVL_iXlinker.EtherCAT_Master_EJxxxx.Beckhoff_EJ3xxx.A_0012_EJ3108_0000_0018.AI_Standard_Channel_1.Status/Limit_1 <-> AI Standard Channel 1/Status/Limit 1
//     PlcTask Inputs/GVL_iXlinker.EtherCAT_Master_EJxxxx.Beckhoff_EJ3xxx.A_0012_EJ3108_0000_0018.AI_Standard_Channel_1.Status/Limit_2 <-> AI Standard Channel 1/Status/Limit 2
//     PlcTask Inputs/GVL_iXlinker.EtherCAT_Master_EJxxxx.Beckhoff_EJ3xxx.A_0012_EJ3108_0000_0018.AI_Standard_Channel_2.Status/Limit_1 <-> AI Standard Channel 2/Status/Limit 1
//     PlcTask Inputs/GVL_iXlinker.EtherCAT_Master_EJxxxx.Beckhoff_EJ3xxx.A_0012_EJ3108_0000_0018.AI_Standard_Channel_2.Status/Limit_2 <-> AI Standard Channel 2/Status/Limit 2
//     PlcTask Inputs/GVL_iXlinker.EtherCAT_Master_EJxxxx.Beckhoff_EJ3xxx.A_0012_EJ3108_0000_0018.AI_Standard_Channel_3.Status/Limit_1 <-> AI Standard Channel 3/Status/Limit 1
//     PlcTask Inputs/GVL_iXlinker.EtherCAT_Master_EJxxxx.Beckhoff_EJ3xxx.A_0012_EJ3108_0000_0018.AI_Standard_Channel_3.Status/Limit_2 <-> AI Standard Channel 3/Status/Limit 2
//     PlcTask Inputs/GVL_iXlinker.EtherCAT_Master_EJxxxx.Beckhoff_EJ3xxx.A_0012_EJ3108_0000_0018.AI_Standard_Channel_4.Status/Limit_1 <-> AI Standard Channel 4/Status/Limit 1
//     PlcTask Inputs/GVL_iXlinker.EtherCAT_Master_EJxxxx.Beckhoff_EJ3xxx.A_0012_EJ3108_0000_0018.AI_Standard_Channel_4.Status/Limit_2 <-> AI Standard Channel 4/Status/Limit 2
//     PlcTask Inputs/GVL_iXlinker.EtherCAT_Master_EJxxxx.Beckhoff_EJ3xxx.A_0012_EJ3108_0000_0018.AI_Standard_Channel_5.Status/Limit_1 <-> AI Standard Channel 5/Status/Limit 1
//     PlcTask Inputs/GVL_iXlinker.EtherCAT_Master_EJxxxx.Beckhoff_EJ3xxx.A_0012_EJ3108_0000_0018.AI_Standard_Channel_5.Status/Limit_2 <-> AI Standard Channel 5/Status/Limit 2
//     PlcTask Inputs/GVL_iXlinker.EtherCAT_Master_EJxxxx.Beckhoff_EJ3xxx.A_0012_EJ3108_0000_0018.AI_Standard_Channel_6.Status/Limit_1 <-> AI Standard Channel 6/Status/Limit 1
//     PlcTask Inputs/GVL_iXlinker.EtherCAT_Master_EJxxxx.Beckhoff_EJ3xxx.A_0012_EJ3108_0000_0018.AI_Standard_Channel_6.Status/Limit_2 <-> AI Standard Channel 6/Status/Limit 2
//     PlcTask Inputs/GVL_iXlinker.EtherCAT_Master_EJxxxx.Beckhoff_EJ3xxx.A_0012_EJ3108_0000_0018.AI_Standard_Channel_7.Status/Limit_1 <-> AI Standard Channel 7/Status/Limit 1
//     PlcTask Inputs/GVL_iXlinker.EtherCAT_Master_EJxxxx.Beckhoff_EJ3xxx.A_0012_EJ3108_0000_0018.AI_Standard_Channel_7.Status/Limit_2 <-> AI Standard Channel 7/Status/Limit 2
//     PlcTask Inputs/GVL_iXlinker.EtherCAT_Master_EJxxxx.Beckhoff_EJ3xxx.A_0012_EJ3108_0000_0018.AI_Standard_Channel_8.Status/Limit_1 <-> AI Standard Channel 8/Status/Limit 1
//     PlcTask Inputs/GVL_iXlinker.EtherCAT_Master_EJxxxx.Beckhoff_EJ3xxx.A_0012_EJ3108_0000_0018.AI_Standard_Channel_8.Status/Limit_2 <-> AI Standard Channel 8/Status/Limit 2
//     PlcTask Inputs/GVL_iXlinker.EtherCAT_Master_EJxxxx.Beckhoff_EJ3xxx.A_0012_EJ3108_0000_0018.AI_Standard_Channel_1.Status/Error <-> AI Standard Channel 1/Status/Error
//     PlcTask Inputs/GVL_iXlinker.EtherCAT_Master_EJxxxx.Beckhoff_EJ3xxx.A_0012_EJ3108_0000_0018.AI_Standard_Channel_2.Status/Error <-> AI Standard Channel 2/Status/Error
//     PlcTask Inputs/GVL_iXlinker.EtherCAT_Master_EJxxxx.Beckhoff_EJ3xxx.A_0012_EJ3108_0000_0018.AI_Standard_Channel_3.Status/Error <-> AI Standard Channel 3/Status/Error
//     PlcTask Inputs/GVL_iXlinker.EtherCAT_Master_EJxxxx.Beckhoff_EJ3xxx.A_0012_EJ3108_0000_0018.AI_Standard_Channel_4.Status/Error <-> AI Standard Channel 4/Status/Error
//     PlcTask Inputs/GVL_iXlinker.EtherCAT_Master_EJxxxx.Beckhoff_EJ3xxx.A_0012_EJ3108_0000_0018.AI_Standard_Channel_5.Status/Error <-> AI Standard Channel 5/Status/Error
//     PlcTask Inputs/GVL_iXlinker.EtherCAT_Master_EJxxxx.Beckhoff_EJ3xxx.A_0012_EJ3108_0000_0018.AI_Standard_Channel_6.Status/Error <-> AI Standard Channel 6/Status/Error
//     PlcTask Inputs/GVL_iXlinker.EtherCAT_Master_EJxxxx.Beckhoff_EJ3xxx.A_0012_EJ3108_0000_0018.AI_Standard_Channel_7.Status/Error <-> AI Standard Channel 7/Status/Error
//     PlcTask Inputs/GVL_iXlinker.EtherCAT_Master_EJxxxx.Beckhoff_EJ3xxx.A_0012_EJ3108_0000_0018.AI_Standard_Channel_8.Status/Error <-> AI Standard Channel 8/Status/Error
//     PlcTask Inputs/GVL_iXlinker.EtherCAT_Master_EJxxxx.Beckhoff_EJ3xxx.A_0012_EJ3108_0000_0018.AI_Standard_Channel_1.Status/Sync_error <-> AI Standard Channel 1/Status/Sync error
//     PlcTask Inputs/GVL_iXlinker.EtherCAT_Master_EJxxxx.Beckhoff_EJ3xxx.A_0012_EJ3108_0000_0018.AI_Standard_Channel_2.Status/Sync_error <-> AI Standard Channel 2/Status/Sync error
//     PlcTask Inputs/GVL_iXlinker.EtherCAT_Master_EJxxxx.Beckhoff_EJ3xxx.A_0012_EJ3108_0000_0018.AI_Standard_Channel_3.Status/Sync_error <-> AI Standard Channel 3/Status/Sync error
//     PlcTask Inputs/GVL_iXlinker.EtherCAT_Master_EJxxxx.Beckhoff_EJ3xxx.A_0012_EJ3108_0000_0018.AI_Standard_Channel_4.Status/Sync_error <-> AI Standard Channel 4/Status/Sync error
//     PlcTask Inputs/GVL_iXlinker.EtherCAT_Master_EJxxxx.Beckhoff_EJ3xxx.A_0012_EJ3108_0000_0018.AI_Standard_Channel_5.Status/Sync_error <-> AI Standard Channel 5/Status/Sync error
//     PlcTask Inputs/GVL_iXlinker.EtherCAT_Master_EJxxxx.Beckhoff_EJ3xxx.A_0012_EJ3108_0000_0018.AI_Standard_Channel_6.Status/Sync_error <-> AI Standard Channel 6/Status/Sync error
//     PlcTask Inputs/GVL_iXlinker.EtherCAT_Master_EJxxxx.Beckhoff_EJ3xxx.A_0012_EJ3108_0000_0018.AI_Standard_Channel_7.Status/Sync_error <-> AI Standard Channel 7/Status/Sync error
//     PlcTask Inputs/GVL_iXlinker.EtherCAT_Master_EJxxxx.Beckhoff_EJ3xxx.A_0012_EJ3108_0000_0018.AI_Standard_Channel_8.Status/Sync_error <-> AI Standard Channel 8/Status/Sync error
//     PlcTask Inputs/GVL_iXlinker.EtherCAT_Master_EJxxxx.Beckhoff_EJ3xxx.A_0012_EJ3108_0000_0018.AI_Standard_Channel_1.Status/TxPDO_State <-> AI Standard Channel 1/Status/TxPDO State
//     PlcTask Inputs/GVL_iXlinker.EtherCAT_Master_EJxxxx.Beckhoff_EJ3xxx.A_0012_EJ3108_0000_0018.AI_Standard_Channel_2.Status/TxPDO_State <-> AI Standard Channel 2/Status/TxPDO State
//     PlcTask Inputs/GVL_iXlinker.EtherCAT_Master_EJxxxx.Beckhoff_EJ3xxx.A_0012_EJ3108_0000_0018.AI_Standard_Channel_3.Status/TxPDO_State <-> AI Standard Channel 3/Status/TxPDO State
//     PlcTask Inputs/GVL_iXlinker.EtherCAT_Master_EJxxxx.Beckhoff_EJ3xxx.A_0012_EJ3108_0000_0018.AI_Standard_Channel_4.Status/TxPDO_State <-> AI Standard Channel 4/Status/TxPDO State
//     PlcTask Inputs/GVL_iXlinker.EtherCAT_Master_EJxxxx.Beckhoff_EJ3xxx.A_0012_EJ3108_0000_0018.AI_Standard_Channel_5.Status/TxPDO_State <-> AI Standard Channel 5/Status/TxPDO State
//     PlcTask Inputs/GVL_iXlinker.EtherCAT_Master_EJxxxx.Beckhoff_EJ3xxx.A_0012_EJ3108_0000_0018.AI_Standard_Channel_6.Status/TxPDO_State <-> AI Standard Channel 6/Status/TxPDO State
//     PlcTask Inputs/GVL_iXlinker.EtherCAT_Master_EJxxxx.Beckhoff_EJ3xxx.A_0012_EJ3108_0000_0018.AI_Standard_Channel_7.Status/TxPDO_State <-> AI Standard Channel 7/Status/TxPDO State
//     PlcTask Inputs/GVL_iXlinker.EtherCAT_Master_EJxxxx.Beckhoff_EJ3xxx.A_0012_EJ3108_0000_0018.AI_Standard_Channel_8.Status/TxPDO_State <-> AI Standard Channel 8/Status/TxPDO State
//     PlcTask Inputs/GVL_iXlinker.EtherCAT_Master_EJxxxx.Beckhoff_EJ3xxx.A_0012_EJ3108_0000_0018.AI_Standard_Channel_1.Status/TxPDO_Toggle <-> AI Standard Channel 1/Status/TxPDO Toggle
//     PlcTask Inputs/GVL_iXlinker.EtherCAT_Master_EJxxxx.Beckhoff_EJ3xxx.A_0012_EJ3108_0000_0018.AI_Standard_Channel_2.Status/TxPDO_Toggle <-> AI Standard Channel 2/Status/TxPDO Toggle
//     PlcTask Inputs/GVL_iXlinker.EtherCAT_Master_EJxxxx.Beckhoff_EJ3xxx.A_0012_EJ3108_0000_0018.AI_Standard_Channel_3.Status/TxPDO_Toggle <-> AI Standard Channel 3/Status/TxPDO Toggle
//     PlcTask Inputs/GVL_iXlinker.EtherCAT_Master_EJxxxx.Beckhoff_EJ3xxx.A_0012_EJ3108_0000_0018.AI_Standard_Channel_4.Status/TxPDO_Toggle <-> AI Standard Channel 4/Status/TxPDO Toggle
//     PlcTask Inputs/GVL_iXlinker.EtherCAT_Master_EJxxxx.Beckhoff_EJ3xxx.A_0012_EJ3108_0000_0018.AI_Standard_Channel_5.Status/TxPDO_Toggle <-> AI Standard Channel 5/Status/TxPDO Toggle
//     PlcTask Inputs/GVL_iXlinker.EtherCAT_Master_EJxxxx.Beckhoff_EJ3xxx.A_0012_EJ3108_0000_0018.AI_Standard_Channel_6.Status/TxPDO_Toggle <-> AI Standard Channel 6/Status/TxPDO Toggle
//     PlcTask Inputs/GVL_iXlinker.EtherCAT_Master_EJxxxx.Beckhoff_EJ3xxx.A_0012_EJ3108_0000_0018.AI_Standard_Channel_7.Status/TxPDO_Toggle <-> AI Standard Channel 7/Status/TxPDO Toggle
//     PlcTask Inputs/GVL_iXlinker.EtherCAT_Master_EJxxxx.Beckhoff_EJ3xxx.A_0012_EJ3108_0000_0018.AI_Standard_Channel_8.Status/TxPDO_Toggle <-> AI Standard Channel 8/Status/TxPDO Toggle
//     PlcTask Inputs/GVL_iXlinker.EtherCAT_Master_EJxxxx.Beckhoff_EJ3xxx.A_0012_EJ3108_0000_0018.AI_Standard_Channel_1.Value <-> AI Standard Channel 1/Value
//     PlcTask Inputs/GVL_iXlinker.EtherCAT_Master_EJxxxx.Beckhoff_EJ3xxx.A_0012_EJ3108_0000_0018.AI_Standard_Channel_2.Value <-> AI Standard Channel 2/Value
//     PlcTask Inputs/GVL_iXlinker.EtherCAT_Master_EJxxxx.Beckhoff_EJ3xxx.A_0012_EJ3108_0000_0018.AI_Standard_Channel_3.Value <-> AI Standard Channel 3/Value
//     PlcTask Inputs/GVL_iXlinker.EtherCAT_Master_EJxxxx.Beckhoff_EJ3xxx.A_0012_EJ3108_0000_0018.AI_Standard_Channel_4.Value <-> AI Standard Channel 4/Value
//     PlcTask Inputs/GVL_iXlinker.EtherCAT_Master_EJxxxx.Beckhoff_EJ3xxx.A_0012_EJ3108_0000_0018.AI_Standard_Channel_5.Value <-> AI Standard Channel 5/Value
//     PlcTask Inputs/GVL_iXlinker.EtherCAT_Master_EJxxxx.Beckhoff_EJ3xxx.A_0012_EJ3108_0000_0018.AI_Standard_Channel_6.Value <-> AI Standard Channel 6/Value
//     PlcTask Inputs/GVL_iXlinker.EtherCAT_Master_EJxxxx.Beckhoff_EJ3xxx.A_0012_EJ3108_0000_0018.AI_Standard_Channel_7.Value <-> AI Standard Channel 7/Value
//     PlcTask Inputs/GVL_iXlinker.EtherCAT_Master_EJxxxx.Beckhoff_EJ3xxx.A_0012_EJ3108_0000_0018.AI_Standard_Channel_8.Value <-> AI Standard Channel 8/Value
//     PlcTask Inputs/GVL_iXlinker.EtherCAT_Master_EJxxxx.Beckhoff_EJ3xxx.A_0012_EJ3108_0000_0018.WcState.WcState <-> WcState/WcState
//     PlcTask Inputs/GVL_iXlinker.EtherCAT_Master_EJxxxx.Beckhoff_EJ3xxx.A_0012_EJ3108_0000_0018.WcState.InputToggle <-> WcState/InputToggle
//     PlcTask Inputs/GVL_iXlinker.EtherCAT_Master_EJxxxx.Beckhoff_EJ3xxx.A_0012_EJ3108_0000_0018.InfoData.AdsAddr <-> InfoData/AdsAddr
//     PlcTask Inputs/GVL_iXlinker.EtherCAT_Master_EJxxxx.Beckhoff_EJ3xxx.A_0012_EJ3108_0000_0018.InfoData.State <-> InfoData/State
//   PLC/PLC Instance <-> EtherCAT Master EJxxxx/Beckhoff EJ3xxx/A_0013(EJ3108-0000-0019)
//     PlcTask Inputs/GVL_iXlinker.EtherCAT_Master_EJxxxx.Beckhoff_EJ3xxx.A_0013_EJ3108_0000_0019.AI_Standard_Channel_1.Status/Underrange <-> AI Standard Channel 1/Status/Underrange
//     PlcTask Inputs/GVL_iXlinker.EtherCAT_Master_EJxxxx.Beckhoff_EJ3xxx.A_0013_EJ3108_0000_0019.AI_Standard_Channel_2.Status/Underrange <-> AI Standard Channel 2/Status/Underrange
//     PlcTask Inputs/GVL_iXlinker.EtherCAT_Master_EJxxxx.Beckhoff_EJ3xxx.A_0013_EJ3108_0000_0019.AI_Standard_Channel_3.Status/Underrange <-> AI Standard Channel 3/Status/Underrange
//     PlcTask Inputs/GVL_iXlinker.EtherCAT_Master_EJxxxx.Beckhoff_EJ3xxx.A_0013_EJ3108_0000_0019.AI_Standard_Channel_4.Status/Underrange <-> AI Standard Channel 4/Status/Underrange
//     PlcTask Inputs/GVL_iXlinker.EtherCAT_Master_EJxxxx.Beckhoff_EJ3xxx.A_0013_EJ3108_0000_0019.AI_Standard_Channel_5.Status/Underrange <-> AI Standard Channel 5/Status/Underrange
//     PlcTask Inputs/GVL_iXlinker.EtherCAT_Master_EJxxxx.Beckhoff_EJ3xxx.A_0013_EJ3108_0000_0019.AI_Standard_Channel_6.Status/Underrange <-> AI Standard Channel 6/Status/Underrange
//     PlcTask Inputs/GVL_iXlinker.EtherCAT_Master_EJxxxx.Beckhoff_EJ3xxx.A_0013_EJ3108_0000_0019.AI_Standard_Channel_7.Status/Underrange <-> AI Standard Channel 7/Status/Underrange
//     PlcTask Inputs/GVL_iXlinker.EtherCAT_Master_EJxxxx.Beckhoff_EJ3xxx.A_0013_EJ3108_0000_0019.AI_Standard_Channel_8.Status/Underrange <-> AI Standard Channel 8/Status/Underrange
//     PlcTask Inputs/GVL_iXlinker.EtherCAT_Master_EJxxxx.Beckhoff_EJ3xxx.A_0013_EJ3108_0000_0019.AI_Standard_Channel_1.Status/Overrange <-> AI Standard Channel 1/Status/Overrange
//     PlcTask Inputs/GVL_iXlinker.EtherCAT_Master_EJxxxx.Beckhoff_EJ3xxx.A_0013_EJ3108_0000_0019.AI_Standard_Channel_2.Status/Overrange <-> AI Standard Channel 2/Status/Overrange
//     PlcTask Inputs/GVL_iXlinker.EtherCAT_Master_EJxxxx.Beckhoff_EJ3xxx.A_0013_EJ3108_0000_0019.AI_Standard_Channel_3.Status/Overrange <-> AI Standard Channel 3/Status/Overrange
//     PlcTask Inputs/GVL_iXlinker.EtherCAT_Master_EJxxxx.Beckhoff_EJ3xxx.A_0013_EJ3108_0000_0019.AI_Standard_Channel_4.Status/Overrange <-> AI Standard Channel 4/Status/Overrange
//     PlcTask Inputs/GVL_iXlinker.EtherCAT_Master_EJxxxx.Beckhoff_EJ3xxx.A_0013_EJ3108_0000_0019.AI_Standard_Channel_5.Status/Overrange <-> AI Standard Channel 5/Status/Overrange
//     PlcTask Inputs/GVL_iXlinker.EtherCAT_Master_EJxxxx.Beckhoff_EJ3xxx.A_0013_EJ3108_0000_0019.AI_Standard_Channel_6.Status/Overrange <-> AI Standard Channel 6/Status/Overrange
//     PlcTask Inputs/GVL_iXlinker.EtherCAT_Master_EJxxxx.Beckhoff_EJ3xxx.A_0013_EJ3108_0000_0019.AI_Standard_Channel_7.Status/Overrange <-> AI Standard Channel 7/Status/Overrange
//     PlcTask Inputs/GVL_iXlinker.EtherCAT_Master_EJxxxx.Beckhoff_EJ3xxx.A_0013_EJ3108_0000_0019.AI_Standard_Channel_8.Status/Overrange <-> AI Standard Channel 8/Status/Overrange
//     PlcTask Inputs/GVL_iXlinker.EtherCAT_Master_EJxxxx.Beckhoff_EJ3xxx.A_0013_EJ3108_0000_0019.AI_Standard_Channel_1.Status/Limit_1 <-> AI Standard Channel 1/Status/Limit 1
//     PlcTask Inputs/GVL_iXlinker.EtherCAT_Master_EJxxxx.Beckhoff_EJ3xxx.A_0013_EJ3108_0000_0019.AI_Standard_Channel_1.Status/Limit_2 <-> AI Standard Channel 1/Status/Limit 2
//     PlcTask Inputs/GVL_iXlinker.EtherCAT_Master_EJxxxx.Beckhoff_EJ3xxx.A_0013_EJ3108_0000_0019.AI_Standard_Channel_2.Status/Limit_1 <-> AI Standard Channel 2/Status/Limit 1
//     PlcTask Inputs/GVL_iXlinker.EtherCAT_Master_EJxxxx.Beckhoff_EJ3xxx.A_0013_EJ3108_0000_0019.AI_Standard_Channel_2.Status/Limit_2 <-> AI Standard Channel 2/Status/Limit 2
//     PlcTask Inputs/GVL_iXlinker.EtherCAT_Master_EJxxxx.Beckhoff_EJ3xxx.A_0013_EJ3108_0000_0019.AI_Standard_Channel_3.Status/Limit_1 <-> AI Standard Channel 3/Status/Limit 1
//     PlcTask Inputs/GVL_iXlinker.EtherCAT_Master_EJxxxx.Beckhoff_EJ3xxx.A_0013_EJ3108_0000_0019.AI_Standard_Channel_3.Status/Limit_2 <-> AI Standard Channel 3/Status/Limit 2
//     PlcTask Inputs/GVL_iXlinker.EtherCAT_Master_EJxxxx.Beckhoff_EJ3xxx.A_0013_EJ3108_0000_0019.AI_Standard_Channel_4.Status/Limit_1 <-> AI Standard Channel 4/Status/Limit 1
//     PlcTask Inputs/GVL_iXlinker.EtherCAT_Master_EJxxxx.Beckhoff_EJ3xxx.A_0013_EJ3108_0000_0019.AI_Standard_Channel_4.Status/Limit_2 <-> AI Standard Channel 4/Status/Limit 2
//     PlcTask Inputs/GVL_iXlinker.EtherCAT_Master_EJxxxx.Beckhoff_EJ3xxx.A_0013_EJ3108_0000_0019.AI_Standard_Channel_5.Status/Limit_1 <-> AI Standard Channel 5/Status/Limit 1
//     PlcTask Inputs/GVL_iXlinker.EtherCAT_Master_EJxxxx.Beckhoff_EJ3xxx.A_0013_EJ3108_0000_0019.AI_Standard_Channel_5.Status/Limit_2 <-> AI Standard Channel 5/Status/Limit 2
//     PlcTask Inputs/GVL_iXlinker.EtherCAT_Master_EJxxxx.Beckhoff_EJ3xxx.A_0013_EJ3108_0000_0019.AI_Standard_Channel_6.Status/Limit_1 <-> AI Standard Channel 6/Status/Limit 1
//     PlcTask Inputs/GVL_iXlinker.EtherCAT_Master_EJxxxx.Beckhoff_EJ3xxx.A_0013_EJ3108_0000_0019.AI_Standard_Channel_6.Status/Limit_2 <-> AI Standard Channel 6/Status/Limit 2
//     PlcTask Inputs/GVL_iXlinker.EtherCAT_Master_EJxxxx.Beckhoff_EJ3xxx.A_0013_EJ3108_0000_0019.AI_Standard_Channel_7.Status/Limit_1 <-> AI Standard Channel 7/Status/Limit 1
//     PlcTask Inputs/GVL_iXlinker.EtherCAT_Master_EJxxxx.Beckhoff_EJ3xxx.A_0013_EJ3108_0000_0019.AI_Standard_Channel_7.Status/Limit_2 <-> AI Standard Channel 7/Status/Limit 2
//     PlcTask Inputs/GVL_iXlinker.EtherCAT_Master_EJxxxx.Beckhoff_EJ3xxx.A_0013_EJ3108_0000_0019.AI_Standard_Channel_8.Status/Limit_1 <-> AI Standard Channel 8/Status/Limit 1
//     PlcTask Inputs/GVL_iXlinker.EtherCAT_Master_EJxxxx.Beckhoff_EJ3xxx.A_0013_EJ3108_0000_0019.AI_Standard_Channel_8.Status/Limit_2 <-> AI Standard Channel 8/Status/Limit 2
//     PlcTask Inputs/GVL_iXlinker.EtherCAT_Master_EJxxxx.Beckhoff_EJ3xxx.A_0013_EJ3108_0000_0019.AI_Standard_Channel_1.Status/Error <-> AI Standard Channel 1/Status/Error
//     PlcTask Inputs/GVL_iXlinker.EtherCAT_Master_EJxxxx.Beckhoff_EJ3xxx.A_0013_EJ3108_0000_0019.AI_Standard_Channel_2.Status/Error <-> AI Standard Channel 2/Status/Error
//     PlcTask Inputs/GVL_iXlinker.EtherCAT_Master_EJxxxx.Beckhoff_EJ3xxx.A_0013_EJ3108_0000_0019.AI_Standard_Channel_3.Status/Error <-> AI Standard Channel 3/Status/Error
//     PlcTask Inputs/GVL_iXlinker.EtherCAT_Master_EJxxxx.Beckhoff_EJ3xxx.A_0013_EJ3108_0000_0019.AI_Standard_Channel_4.Status/Error <-> AI Standard Channel 4/Status/Error
//     PlcTask Inputs/GVL_iXlinker.EtherCAT_Master_EJxxxx.Beckhoff_EJ3xxx.A_0013_EJ3108_0000_0019.AI_Standard_Channel_5.Status/Error <-> AI Standard Channel 5/Status/Error
//     PlcTask Inputs/GVL_iXlinker.EtherCAT_Master_EJxxxx.Beckhoff_EJ3xxx.A_0013_EJ3108_0000_0019.AI_Standard_Channel_6.Status/Error <-> AI Standard Channel 6/Status/Error
//     PlcTask Inputs/GVL_iXlinker.EtherCAT_Master_EJxxxx.Beckhoff_EJ3xxx.A_0013_EJ3108_0000_0019.AI_Standard_Channel_7.Status/Error <-> AI Standard Channel 7/Status/Error
//     PlcTask Inputs/GVL_iXlinker.EtherCAT_Master_EJxxxx.Beckhoff_EJ3xxx.A_0013_EJ3108_0000_0019.AI_Standard_Channel_8.Status/Error <-> AI Standard Channel 8/Status/Error
//     PlcTask Inputs/GVL_iXlinker.EtherCAT_Master_EJxxxx.Beckhoff_EJ3xxx.A_0013_EJ3108_0000_0019.AI_Standard_Channel_1.Status/Sync_error <-> AI Standard Channel 1/Status/Sync error
//     PlcTask Inputs/GVL_iXlinker.EtherCAT_Master_EJxxxx.Beckhoff_EJ3xxx.A_0013_EJ3108_0000_0019.AI_Standard_Channel_2.Status/Sync_error <-> AI Standard Channel 2/Status/Sync error
//     PlcTask Inputs/GVL_iXlinker.EtherCAT_Master_EJxxxx.Beckhoff_EJ3xxx.A_0013_EJ3108_0000_0019.AI_Standard_Channel_3.Status/Sync_error <-> AI Standard Channel 3/Status/Sync error
//     PlcTask Inputs/GVL_iXlinker.EtherCAT_Master_EJxxxx.Beckhoff_EJ3xxx.A_0013_EJ3108_0000_0019.AI_Standard_Channel_4.Status/Sync_error <-> AI Standard Channel 4/Status/Sync error
//     PlcTask Inputs/GVL_iXlinker.EtherCAT_Master_EJxxxx.Beckhoff_EJ3xxx.A_0013_EJ3108_0000_0019.AI_Standard_Channel_5.Status/Sync_error <-> AI Standard Channel 5/Status/Sync error
//     PlcTask Inputs/GVL_iXlinker.EtherCAT_Master_EJxxxx.Beckhoff_EJ3xxx.A_0013_EJ3108_0000_0019.AI_Standard_Channel_6.Status/Sync_error <-> AI Standard Channel 6/Status/Sync error
//     PlcTask Inputs/GVL_iXlinker.EtherCAT_Master_EJxxxx.Beckhoff_EJ3xxx.A_0013_EJ3108_0000_0019.AI_Standard_Channel_7.Status/Sync_error <-> AI Standard Channel 7/Status/Sync error
//     PlcTask Inputs/GVL_iXlinker.EtherCAT_Master_EJxxxx.Beckhoff_EJ3xxx.A_0013_EJ3108_0000_0019.AI_Standard_Channel_8.Status/Sync_error <-> AI Standard Channel 8/Status/Sync error
//     PlcTask Inputs/GVL_iXlinker.EtherCAT_Master_EJxxxx.Beckhoff_EJ3xxx.A_0013_EJ3108_0000_0019.AI_Standard_Channel_1.Status/TxPDO_State <-> AI Standard Channel 1/Status/TxPDO State
//     PlcTask Inputs/GVL_iXlinker.EtherCAT_Master_EJxxxx.Beckhoff_EJ3xxx.A_0013_EJ3108_0000_0019.AI_Standard_Channel_2.Status/TxPDO_State <-> AI Standard Channel 2/Status/TxPDO State
//     PlcTask Inputs/GVL_iXlinker.EtherCAT_Master_EJxxxx.Beckhoff_EJ3xxx.A_0013_EJ3108_0000_0019.AI_Standard_Channel_3.Status/TxPDO_State <-> AI Standard Channel 3/Status/TxPDO State
//     PlcTask Inputs/GVL_iXlinker.EtherCAT_Master_EJxxxx.Beckhoff_EJ3xxx.A_0013_EJ3108_0000_0019.AI_Standard_Channel_4.Status/TxPDO_State <-> AI Standard Channel 4/Status/TxPDO State
//     PlcTask Inputs/GVL_iXlinker.EtherCAT_Master_EJxxxx.Beckhoff_EJ3xxx.A_0013_EJ3108_0000_0019.AI_Standard_Channel_5.Status/TxPDO_State <-> AI Standard Channel 5/Status/TxPDO State
//     PlcTask Inputs/GVL_iXlinker.EtherCAT_Master_EJxxxx.Beckhoff_EJ3xxx.A_0013_EJ3108_0000_0019.AI_Standard_Channel_6.Status/TxPDO_State <-> AI Standard Channel 6/Status/TxPDO State
//     PlcTask Inputs/GVL_iXlinker.EtherCAT_Master_EJxxxx.Beckhoff_EJ3xxx.A_0013_EJ3108_0000_0019.AI_Standard_Channel_7.Status/TxPDO_State <-> AI Standard Channel 7/Status/TxPDO State
//     PlcTask Inputs/GVL_iXlinker.EtherCAT_Master_EJxxxx.Beckhoff_EJ3xxx.A_0013_EJ3108_0000_0019.AI_Standard_Channel_8.Status/TxPDO_State <-> AI Standard Channel 8/Status/TxPDO State
//     PlcTask Inputs/GVL_iXlinker.EtherCAT_Master_EJxxxx.Beckhoff_EJ3xxx.A_0013_EJ3108_0000_0019.AI_Standard_Channel_1.Status/TxPDO_Toggle <-> AI Standard Channel 1/Status/TxPDO Toggle
//     PlcTask Inputs/GVL_iXlinker.EtherCAT_Master_EJxxxx.Beckhoff_EJ3xxx.A_0013_EJ3108_0000_0019.AI_Standard_Channel_2.Status/TxPDO_Toggle <-> AI Standard Channel 2/Status/TxPDO Toggle
//     PlcTask Inputs/GVL_iXlinker.EtherCAT_Master_EJxxxx.Beckhoff_EJ3xxx.A_0013_EJ3108_0000_0019.AI_Standard_Channel_3.Status/TxPDO_Toggle <-> AI Standard Channel 3/Status/TxPDO Toggle
//     PlcTask Inputs/GVL_iXlinker.EtherCAT_Master_EJxxxx.Beckhoff_EJ3xxx.A_0013_EJ3108_0000_0019.AI_Standard_Channel_4.Status/TxPDO_Toggle <-> AI Standard Channel 4/Status/TxPDO Toggle
//     PlcTask Inputs/GVL_iXlinker.EtherCAT_Master_EJxxxx.Beckhoff_EJ3xxx.A_0013_EJ3108_0000_0019.AI_Standard_Channel_5.Status/TxPDO_Toggle <-> AI Standard Channel 5/Status/TxPDO Toggle
//     PlcTask Inputs/GVL_iXlinker.EtherCAT_Master_EJxxxx.Beckhoff_EJ3xxx.A_0013_EJ3108_0000_0019.AI_Standard_Channel_6.Status/TxPDO_Toggle <-> AI Standard Channel 6/Status/TxPDO Toggle
//     PlcTask Inputs/GVL_iXlinker.EtherCAT_Master_EJxxxx.Beckhoff_EJ3xxx.A_0013_EJ3108_0000_0019.AI_Standard_Channel_7.Status/TxPDO_Toggle <-> AI Standard Channel 7/Status/TxPDO Toggle
//     PlcTask Inputs/GVL_iXlinker.EtherCAT_Master_EJxxxx.Beckhoff_EJ3xxx.A_0013_EJ3108_0000_0019.AI_Standard_Channel_8.Status/TxPDO_Toggle <-> AI Standard Channel 8/Status/TxPDO Toggle
//     PlcTask Inputs/GVL_iXlinker.EtherCAT_Master_EJxxxx.Beckhoff_EJ3xxx.A_0013_EJ3108_0000_0019.AI_Standard_Channel_1.Value <-> AI Standard Channel 1/Value
//     PlcTask Inputs/GVL_iXlinker.EtherCAT_Master_EJxxxx.Beckhoff_EJ3xxx.A_0013_EJ3108_0000_0019.AI_Standard_Channel_2.Value <-> AI Standard Channel 2/Value
//     PlcTask Inputs/GVL_iXlinker.EtherCAT_Master_EJxxxx.Beckhoff_EJ3xxx.A_0013_EJ3108_0000_0019.AI_Standard_Channel_3.Value <-> AI Standard Channel 3/Value
//     PlcTask Inputs/GVL_iXlinker.EtherCAT_Master_EJxxxx.Beckhoff_EJ3xxx.A_0013_EJ3108_0000_0019.AI_Standard_Channel_4.Value <-> AI Standard Channel 4/Value
//     PlcTask Inputs/GVL_iXlinker.EtherCAT_Master_EJxxxx.Beckhoff_EJ3xxx.A_0013_EJ3108_0000_0019.AI_Standard_Channel_5.Value <-> AI Standard Channel 5/Value
//     PlcTask Inputs/GVL_iXlinker.EtherCAT_Master_EJxxxx.Beckhoff_EJ3xxx.A_0013_EJ3108_0000_0019.AI_Standard_Channel_6.Value <-> AI Standard Channel 6/Value
//     PlcTask Inputs/GVL_iXlinker.EtherCAT_Master_EJxxxx.Beckhoff_EJ3xxx.A_0013_EJ3108_0000_0019.AI_Standard_Channel_7.Value <-> AI Standard Channel 7/Value
//     PlcTask Inputs/GVL_iXlinker.EtherCAT_Master_EJxxxx.Beckhoff_EJ3xxx.A_0013_EJ3108_0000_0019.AI_Standard_Channel_8.Value <-> AI Standard Channel 8/Value
//     PlcTask Inputs/GVL_iXlinker.EtherCAT_Master_EJxxxx.Beckhoff_EJ3xxx.A_0013_EJ3108_0000_0019.WcState.WcState <-> WcState/WcState
//     PlcTask Inputs/GVL_iXlinker.EtherCAT_Master_EJxxxx.Beckhoff_EJ3xxx.A_0013_EJ3108_0000_0019.WcState.InputToggle <-> WcState/InputToggle
//     PlcTask Inputs/GVL_iXlinker.EtherCAT_Master_EJxxxx.Beckhoff_EJ3xxx.A_0013_EJ3108_0000_0019.InfoData.AdsAddr <-> InfoData/AdsAddr
//     PlcTask Inputs/GVL_iXlinker.EtherCAT_Master_EJxxxx.Beckhoff_EJ3xxx.A_0013_EJ3108_0000_0019.InfoData.State <-> InfoData/State
//   PLC/PLC Instance <-> EtherCAT Master EJxxxx/Beckhoff EJ3xxx/A_0014(EJ3202-0000-0019)
//     PlcTask Inputs/GVL_iXlinker.EtherCAT_Master_EJxxxx.Beckhoff_EJ3xxx.A_0014_EJ3202_0000_0019.RTD_Inputs_Channel_1.Status/Underrange <-> RTD Inputs Channel 1/Status/Underrange
//     PlcTask Inputs/GVL_iXlinker.EtherCAT_Master_EJxxxx.Beckhoff_EJ3xxx.A_0014_EJ3202_0000_0019.RTD_Inputs_Channel_2.Status/Underrange <-> RTD Inputs Channel 2/Status/Underrange
//     PlcTask Inputs/GVL_iXlinker.EtherCAT_Master_EJxxxx.Beckhoff_EJ3xxx.A_0014_EJ3202_0000_0019.RTD_Inputs_Channel_1.Status/Overrange <-> RTD Inputs Channel 1/Status/Overrange
//     PlcTask Inputs/GVL_iXlinker.EtherCAT_Master_EJxxxx.Beckhoff_EJ3xxx.A_0014_EJ3202_0000_0019.RTD_Inputs_Channel_2.Status/Overrange <-> RTD Inputs Channel 2/Status/Overrange
//     PlcTask Inputs/GVL_iXlinker.EtherCAT_Master_EJxxxx.Beckhoff_EJ3xxx.A_0014_EJ3202_0000_0019.RTD_Inputs_Channel_1.Status/Limit_1 <-> RTD Inputs Channel 1/Status/Limit 1
//     PlcTask Inputs/GVL_iXlinker.EtherCAT_Master_EJxxxx.Beckhoff_EJ3xxx.A_0014_EJ3202_0000_0019.RTD_Inputs_Channel_1.Status/Limit_2 <-> RTD Inputs Channel 1/Status/Limit 2
//     PlcTask Inputs/GVL_iXlinker.EtherCAT_Master_EJxxxx.Beckhoff_EJ3xxx.A_0014_EJ3202_0000_0019.RTD_Inputs_Channel_2.Status/Limit_1 <-> RTD Inputs Channel 2/Status/Limit 1
//     PlcTask Inputs/GVL_iXlinker.EtherCAT_Master_EJxxxx.Beckhoff_EJ3xxx.A_0014_EJ3202_0000_0019.RTD_Inputs_Channel_2.Status/Limit_2 <-> RTD Inputs Channel 2/Status/Limit 2
//     PlcTask Inputs/GVL_iXlinker.EtherCAT_Master_EJxxxx.Beckhoff_EJ3xxx.A_0014_EJ3202_0000_0019.RTD_Inputs_Channel_1.Status/Error <-> RTD Inputs Channel 1/Status/Error
//     PlcTask Inputs/GVL_iXlinker.EtherCAT_Master_EJxxxx.Beckhoff_EJ3xxx.A_0014_EJ3202_0000_0019.RTD_Inputs_Channel_2.Status/Error <-> RTD Inputs Channel 2/Status/Error
//     PlcTask Inputs/GVL_iXlinker.EtherCAT_Master_EJxxxx.Beckhoff_EJ3xxx.A_0014_EJ3202_0000_0019.RTD_Inputs_Channel_1.Status/TxPDO_State <-> RTD Inputs Channel 1/Status/TxPDO State
//     PlcTask Inputs/GVL_iXlinker.EtherCAT_Master_EJxxxx.Beckhoff_EJ3xxx.A_0014_EJ3202_0000_0019.RTD_Inputs_Channel_2.Status/TxPDO_State <-> RTD Inputs Channel 2/Status/TxPDO State
//     PlcTask Inputs/GVL_iXlinker.EtherCAT_Master_EJxxxx.Beckhoff_EJ3xxx.A_0014_EJ3202_0000_0019.RTD_Inputs_Channel_1.Status/TxPDO_Toggle <-> RTD Inputs Channel 1/Status/TxPDO Toggle
//     PlcTask Inputs/GVL_iXlinker.EtherCAT_Master_EJxxxx.Beckhoff_EJ3xxx.A_0014_EJ3202_0000_0019.RTD_Inputs_Channel_2.Status/TxPDO_Toggle <-> RTD Inputs Channel 2/Status/TxPDO Toggle
//     PlcTask Inputs/GVL_iXlinker.EtherCAT_Master_EJxxxx.Beckhoff_EJ3xxx.A_0014_EJ3202_0000_0019.RTD_Inputs_Channel_1.Value <-> RTD Inputs Channel 1/Value
//     PlcTask Inputs/GVL_iXlinker.EtherCAT_Master_EJxxxx.Beckhoff_EJ3xxx.A_0014_EJ3202_0000_0019.RTD_Inputs_Channel_2.Value <-> RTD Inputs Channel 2/Value
//     PlcTask Inputs/GVL_iXlinker.EtherCAT_Master_EJxxxx.Beckhoff_EJ3xxx.A_0014_EJ3202_0000_0019.WcState.WcState <-> WcState/WcState
//     PlcTask Inputs/GVL_iXlinker.EtherCAT_Master_EJxxxx.Beckhoff_EJ3xxx.A_0014_EJ3202_0000_0019.WcState.InputToggle <-> WcState/InputToggle
//     PlcTask Inputs/GVL_iXlinker.EtherCAT_Master_EJxxxx.Beckhoff_EJ3xxx.A_0014_EJ3202_0000_0019.InfoData.AdsAddr <-> InfoData/AdsAddr
//     PlcTask Inputs/GVL_iXlinker.EtherCAT_Master_EJxxxx.Beckhoff_EJ3xxx.A_0014_EJ3202_0000_0019.InfoData.State <-> InfoData/State
//   PLC/PLC Instance <-> EtherCAT Master EJxxxx/Beckhoff EJ3xxx/A_0015(EJ3202-0000-0020)
//     PlcTask Inputs/GVL_iXlinker.EtherCAT_Master_EJxxxx.Beckhoff_EJ3xxx.A_0015_EJ3202_0000_0020.RTD_Inputs_Channel_1.Status/Underrange <-> RTD Inputs Channel 1/Status/Underrange
//     PlcTask Inputs/GVL_iXlinker.EtherCAT_Master_EJxxxx.Beckhoff_EJ3xxx.A_0015_EJ3202_0000_0020.RTD_Inputs_Channel_2.Status/Underrange <-> RTD Inputs Channel 2/Status/Underrange
//     PlcTask Inputs/GVL_iXlinker.EtherCAT_Master_EJxxxx.Beckhoff_EJ3xxx.A_0015_EJ3202_0000_0020.RTD_Inputs_Channel_1.Status/Overrange <-> RTD Inputs Channel 1/Status/Overrange
//     PlcTask Inputs/GVL_iXlinker.EtherCAT_Master_EJxxxx.Beckhoff_EJ3xxx.A_0015_EJ3202_0000_0020.RTD_Inputs_Channel_2.Status/Overrange <-> RTD Inputs Channel 2/Status/Overrange
//     PlcTask Inputs/GVL_iXlinker.EtherCAT_Master_EJxxxx.Beckhoff_EJ3xxx.A_0015_EJ3202_0000_0020.RTD_Inputs_Channel_1.Status/Limit_1 <-> RTD Inputs Channel 1/Status/Limit 1
//     PlcTask Inputs/GVL_iXlinker.EtherCAT_Master_EJxxxx.Beckhoff_EJ3xxx.A_0015_EJ3202_0000_0020.RTD_Inputs_Channel_1.Status/Limit_2 <-> RTD Inputs Channel 1/Status/Limit 2
//     PlcTask Inputs/GVL_iXlinker.EtherCAT_Master_EJxxxx.Beckhoff_EJ3xxx.A_0015_EJ3202_0000_0020.RTD_Inputs_Channel_2.Status/Limit_1 <-> RTD Inputs Channel 2/Status/Limit 1
//     PlcTask Inputs/GVL_iXlinker.EtherCAT_Master_EJxxxx.Beckhoff_EJ3xxx.A_0015_EJ3202_0000_0020.RTD_Inputs_Channel_2.Status/Limit_2 <-> RTD Inputs Channel 2/Status/Limit 2
//     PlcTask Inputs/GVL_iXlinker.EtherCAT_Master_EJxxxx.Beckhoff_EJ3xxx.A_0015_EJ3202_0000_0020.RTD_Inputs_Channel_1.Status/Error <-> RTD Inputs Channel 1/Status/Error
//     PlcTask Inputs/GVL_iXlinker.EtherCAT_Master_EJxxxx.Beckhoff_EJ3xxx.A_0015_EJ3202_0000_0020.RTD_Inputs_Channel_2.Status/Error <-> RTD Inputs Channel 2/Status/Error
//     PlcTask Inputs/GVL_iXlinker.EtherCAT_Master_EJxxxx.Beckhoff_EJ3xxx.A_0015_EJ3202_0000_0020.RTD_Inputs_Channel_1.Status/TxPDO_State <-> RTD Inputs Channel 1/Status/TxPDO State
//     PlcTask Inputs/GVL_iXlinker.EtherCAT_Master_EJxxxx.Beckhoff_EJ3xxx.A_0015_EJ3202_0000_0020.RTD_Inputs_Channel_2.Status/TxPDO_State <-> RTD Inputs Channel 2/Status/TxPDO State
//     PlcTask Inputs/GVL_iXlinker.EtherCAT_Master_EJxxxx.Beckhoff_EJ3xxx.A_0015_EJ3202_0000_0020.RTD_Inputs_Channel_1.Status/TxPDO_Toggle <-> RTD Inputs Channel 1/Status/TxPDO Toggle
//     PlcTask Inputs/GVL_iXlinker.EtherCAT_Master_EJxxxx.Beckhoff_EJ3xxx.A_0015_EJ3202_0000_0020.RTD_Inputs_Channel_2.Status/TxPDO_Toggle <-> RTD Inputs Channel 2/Status/TxPDO Toggle
//     PlcTask Inputs/GVL_iXlinker.EtherCAT_Master_EJxxxx.Beckhoff_EJ3xxx.A_0015_EJ3202_0000_0020.RTD_Inputs_Channel_1.Value <-> RTD Inputs Channel 1/Value
//     PlcTask Inputs/GVL_iXlinker.EtherCAT_Master_EJxxxx.Beckhoff_EJ3xxx.A_0015_EJ3202_0000_0020.RTD_Inputs_Channel_2.Value <-> RTD Inputs Channel 2/Value
//     PlcTask Inputs/GVL_iXlinker.EtherCAT_Master_EJxxxx.Beckhoff_EJ3xxx.A_0015_EJ3202_0000_0020.WcState.WcState <-> WcState/WcState
//     PlcTask Inputs/GVL_iXlinker.EtherCAT_Master_EJxxxx.Beckhoff_EJ3xxx.A_0015_EJ3202_0000_0020.WcState.InputToggle <-> WcState/InputToggle
//     PlcTask Inputs/GVL_iXlinker.EtherCAT_Master_EJxxxx.Beckhoff_EJ3xxx.A_0015_EJ3202_0000_0020.InfoData.AdsAddr <-> InfoData/AdsAddr
//     PlcTask Inputs/GVL_iXlinker.EtherCAT_Master_EJxxxx.Beckhoff_EJ3xxx.A_0015_EJ3202_0000_0020.InfoData.State <-> InfoData/State
//   PLC/PLC Instance <-> EtherCAT Master EJxxxx/Beckhoff EJ3xxx/A_0016(EJ3202-0000-0021)
//     PlcTask Inputs/GVL_iXlinker.EtherCAT_Master_EJxxxx.Beckhoff_EJ3xxx.A_0016_EJ3202_0000_0021.RTD_Inputs_Channel_1.Status/Underrange <-> RTD Inputs Channel 1/Status/Underrange
//     PlcTask Inputs/GVL_iXlinker.EtherCAT_Master_EJxxxx.Beckhoff_EJ3xxx.A_0016_EJ3202_0000_0021.RTD_Inputs_Channel_2.Status/Underrange <-> RTD Inputs Channel 2/Status/Underrange
//     PlcTask Inputs/GVL_iXlinker.EtherCAT_Master_EJxxxx.Beckhoff_EJ3xxx.A_0016_EJ3202_0000_0021.RTD_Inputs_Channel_1.Status/Overrange <-> RTD Inputs Channel 1/Status/Overrange
//     PlcTask Inputs/GVL_iXlinker.EtherCAT_Master_EJxxxx.Beckhoff_EJ3xxx.A_0016_EJ3202_0000_0021.RTD_Inputs_Channel_2.Status/Overrange <-> RTD Inputs Channel 2/Status/Overrange
//     PlcTask Inputs/GVL_iXlinker.EtherCAT_Master_EJxxxx.Beckhoff_EJ3xxx.A_0016_EJ3202_0000_0021.RTD_Inputs_Channel_1.Status/Limit_1 <-> RTD Inputs Channel 1/Status/Limit 1
//     PlcTask Inputs/GVL_iXlinker.EtherCAT_Master_EJxxxx.Beckhoff_EJ3xxx.A_0016_EJ3202_0000_0021.RTD_Inputs_Channel_1.Status/Limit_2 <-> RTD Inputs Channel 1/Status/Limit 2
//     PlcTask Inputs/GVL_iXlinker.EtherCAT_Master_EJxxxx.Beckhoff_EJ3xxx.A_0016_EJ3202_0000_0021.RTD_Inputs_Channel_2.Status/Limit_1 <-> RTD Inputs Channel 2/Status/Limit 1
